C07161=1021.143,352.231,-144.972,171.488,49.524,159.785
C07162=1021.135,351.990,-144.936,171.480,49.525,159.784
C07163=1021.128,351.749,-144.900,171.473,49.527,159.783
C07164=1021.121,351.507,-144.863,171.466,49.529,159.782
C07165=1021.113,351.266,-144.827,171.459,49.530,159.781
C07166=1021.105,351.019,-144.788,171.451,49.531,159.781
C07167=1021.097,350.772,-144.751,171.444,49.532,159.780
C07168=1021.090,350.525,-144.714,171.437,49.534,159.779
C07169=1021.083,350.278,-144.676,171.429,49.535,159.778
C07170=1021.075,350.031,-144.639,171.422,49.536,159.777
C07171=1021.067,349.784,-144.602,171.416,49.538,159.777
C07172=1021.060,349.537,-144.565,171.408,49.539,159.776
C07173=1021.052,349.289,-144.528,171.400,49.541,159.775
C07174=1021.045,349.042,-144.490,171.393,49.542,159.774
C07175=1021.037,348.795,-144.454,171.386,49.543,159.773
C07176=1021.030,348.548,-144.416,171.379,49.545,159.772
C07177=1021.022,348.302,-144.379,171.371,49.546,159.772
C07178=1021.015,348.054,-144.342,171.364,49.548,159.771
C07179=1021.008,347.807,-144.305,171.357,49.549,159.770
C07180=1021.000,347.560,-144.268,171.350,49.551,159.769
C07181=1020.993,347.313,-144.230,171.343,49.552,159.768
C07182=1020.985,347.065,-144.194,171.336,49.554,159.768
C07183=1020.977,346.818,-144.157,171.329,49.555,159.767
C07184=1020.970,346.571,-144.120,171.321,49.557,159.766
C07185=1020.962,346.324,-144.083,171.314,49.559,159.765
C07186=1020.954,346.076,-144.047,171.308,49.560,159.765
C07187=1020.947,345.829,-144.010,171.300,49.562,159.764
C07188=1020.939,345.582,-143.973,171.293,49.564,159.763
C07189=1020.931,345.335,-143.936,171.286,49.565,159.763
C07190=1020.925,345.087,-143.900,171.279,49.567,159.762
C07191=1020.917,344.840,-143.863,171.272,49.568,159.761
C07192=1020.910,344.593,-143.826,171.265,49.570,159.760
C07193=1020.903,344.346,-143.790,171.258,49.571,159.760
C07194=1020.895,344.099,-143.753,171.250,49.573,159.759
C07195=1020.888,343.851,-143.716,171.244,49.574,159.758
C07196=1020.880,343.604,-143.680,171.237,49.577,159.758
C07197=1020.873,343.358,-143.644,171.230,49.578,159.757
C07198=1020.866,343.110,-143.607,171.223,49.580,159.756
C07199=1020.858,342.863,-143.571,171.216,49.581,159.755
C07200=1020.850,342.615,-143.534,171.208,49.583,159.755
C07201=1020.843,342.368,-143.498,171.202,49.585,159.754
C07202=1020.836,342.121,-143.461,171.195,49.587,159.753
C07203=1020.828,341.874,-143.425,171.189,49.588,159.753
C07204=1020.821,341.626,-143.388,171.182,49.591,159.752
C07205=1020.814,341.379,-143.352,171.174,49.592,159.751
C07206=1020.807,341.132,-143.316,171.168,49.594,159.751
C07207=1020.799,340.884,-143.280,171.161,49.596,159.750
C07208=1020.792,340.638,-143.244,171.154,49.597,159.749
C07209=1020.785,340.390,-143.207,171.147,49.600,159.749
C07210=1020.778,340.143,-143.171,171.140,49.601,159.748
C07211=1020.770,339.896,-143.135,171.134,49.603,159.747
C07212=1020.762,339.648,-143.099,171.127,49.605,159.747
C07213=1020.755,339.402,-143.063,171.120,49.606,159.746
C07214=1020.749,339.153,-143.027,171.113,49.609,159.745
C07215=1020.742,338.906,-142.991,171.106,49.611,159.745
C07216=1020.734,338.659,-142.955,171.100,49.612,159.744
C07217=1020.726,338.411,-142.918,171.093,49.615,159.744
C07218=1020.719,338.169,-142.883,171.086,49.616,159.743
C07219=1020.712,337.926,-142.848,171.079,49.618,159.742
C07220=1020.705,337.684,-142.814,171.073,49.620,159.742
C07221=1020.698,337.441,-142.778,171.066,49.622,159.741
C07222=1020.691,337.198,-142.743,171.060,49.624,159.741
C07223=1020.683,336.956,-142.708,171.054,49.626,159.740
C07224=1020.676,336.713,-142.673,171.047,49.628,159.740
C07225=1020.669,336.470,-142.638,171.040,49.630,159.739
C07226=1020.662,336.222,-142.602,171.033,49.632,159.738
C07227=1020.655,335.975,-142.566,171.027,49.634,159.738
C07228=1020.648,335.727,-142.531,171.020,49.636,159.737
C07229=1020.641,335.480,-142.495,171.014,49.638,159.737
C07230=1020.634,335.233,-142.460,171.007,49.641,159.736
C07231=1020.626,334.985,-142.424,171.001,49.642,159.736
C07232=1020.619,334.738,-142.388,170.994,49.644,159.735
C07233=1020.612,334.490,-142.353,170.988,49.646,159.734
C07234=1020.605,334.243,-142.317,170.981,49.649,159.734
C07235=1020.598,333.996,-142.282,170.975,49.651,159.733
C07236=1020.591,333.748,-142.246,170.968,49.653,159.733
C07237=1020.584,333.501,-142.211,170.962,49.655,159.732
C07238=1020.577,333.254,-142.176,170.955,49.657,159.732
C07239=1020.570,333.006,-142.140,170.949,49.659,159.731
C07240=1020.562,332.759,-142.105,170.942,49.662,159.731
C07241=1020.555,332.512,-142.070,170.936,49.664,159.730
C07242=1020.548,332.264,-142.034,170.929,49.666,159.730
C07243=1020.541,332.016,-141.999,170.923,49.668,159.729
C07244=1020.533,331.769,-141.964,170.916,49.670,159.729
C07245=1020.527,331.522,-141.929,170.910,49.673,159.728
C07246=1020.520,331.275,-141.894,170.903,49.675,159.728
C07247=1020.512,331.027,-141.859,170.897,49.677,159.727
C07248=1020.505,330.780,-141.824,170.890,49.680,159.727
C07249=1020.498,330.532,-141.789,170.884,49.681,159.726
C07250=1020.491,330.285,-141.754,170.877,49.684,159.726
C07251=1020.484,330.037,-141.718,170.871,49.686,159.725
C07252=1020.476,329.790,-141.684,170.864,49.689,159.725
C07253=1020.470,329.542,-141.649,170.858,49.691,159.724
C07254=1020.463,329.295,-141.614,170.851,49.694,159.724
C07255=1020.455,329.048,-141.579,170.845,49.696,159.723
C07256=1020.449,328.800,-141.545,170.838,49.698,159.723
C07257=1020.442,328.553,-141.509,170.833,49.701,159.723
C07258=1020.435,328.305,-141.474,170.826,49.703,159.722
C07259=1020.427,328.057,-141.439,170.820,49.706,159.722
C07260=1020.421,327.810,-141.404,170.814,49.708,159.721
C07261=1020.414,327.562,-141.370,170.807,49.710,159.721
C07262=1020.407,327.315,-141.335,170.801,49.713,159.720
C07263=1020.400,327.068,-141.300,170.794,49.715,159.720
C07264=1020.393,326.820,-141.265,170.789,49.718,159.719
C07265=1020.387,326.572,-141.231,170.782,49.720,159.719
C07266=1020.379,326.325,-141.196,170.776,49.723,159.719
C07267=1020.372,326.078,-141.162,170.769,49.725,159.718
C07268=1020.365,325.830,-141.127,170.763,49.727,159.718
C07269=1020.358,325.583,-141.093,170.758,49.730,159.717
C07270=1020.351,325.335,-141.059,170.751,49.733,159.717
C07271=1020.343,325.088,-141.025,170.745,49.735,159.717
C07272=1020.337,324.840,-140.991,170.738,49.738,159.716
C07273=1020.329,324.593,-140.956,170.733,49.741,159.716
C07274=1020.322,324.345,-140.922,170.726,49.744,159.715
C07275=1020.316,324.097,-140.888,170.720,49.746,159.715
C07276=1020.308,323.850,-140.853,170.713,49.749,159.715
C07277=1020.301,323.602,-140.819,170.708,49.751,159.714
C07278=1020.294,323.357,-140.786,170.701,49.754,159.714
C07279=1020.287,323.112,-140.752,170.695,49.757,159.714
C07280=1020.280,322.867,-140.718,170.689,49.759,159.713
C07281=1020.273,322.622,-140.685,170.683,49.762,159.713
C07282=1020.266,322.377,-140.650,170.677,49.764,159.712
C07283=1020.259,322.132,-140.617,170.671,49.767,159.712
C07284=1020.252,321.888,-140.583,170.665,49.770,159.712
C07285=1020.246,321.642,-140.549,170.659,49.773,159.712
C07286=1020.239,321.395,-140.516,170.653,49.775,159.711
C07287=1020.232,321.147,-140.482,170.647,49.778,159.711
C07288=1020.224,320.899,-140.448,170.641,49.781,159.711
C07289=1020.218,320.651,-140.414,170.634,49.784,159.710
C07290=1020.211,320.405,-140.379,170.629,49.787,159.710
C07291=1020.204,320.157,-140.346,170.623,49.789,159.710
C07292=1020.197,319.909,-140.311,170.616,49.792,159.709
C07293=1020.190,319.661,-140.277,170.611,49.795,159.709
C07294=1020.184,319.415,-140.244,170.604,49.798,159.709
C07295=1020.176,319.167,-140.210,170.598,49.800,159.708
C07296=1020.170,318.918,-140.176,170.593,49.803,159.708
C07297=1020.163,318.671,-140.142,170.586,49.806,159.708
C07298=1020.156,318.424,-140.109,170.580,49.809,159.707
C07299=1020.149,318.176,-140.075,170.574,49.812,159.707
C07300=1020.143,317.928,-140.041,170.568,49.814,159.707
C07301=1020.136,317.681,-140.007,170.563,49.818,159.706
C07302=1020.129,317.433,-139.973,170.556,49.821,159.706
C07303=1020.122,317.186,-139.940,170.551,49.823,159.706
C07304=1020.116,316.938,-139.906,170.545,49.826,159.705
C07305=1020.109,316.690,-139.872,170.538,49.829,159.705
C07306=1020.102,316.443,-139.839,170.533,49.832,159.705
C07307=1020.095,316.195,-139.805,170.527,49.835,159.705
C07308=1020.089,315.947,-139.771,170.521,49.838,159.704
C07309=1020.083,315.700,-139.738,170.515,49.840,159.704
C07310=1020.075,315.452,-139.704,170.510,49.844,159.704
C07311=1020.069,315.205,-139.671,170.503,49.847,159.704
C07312=1020.063,314.957,-139.637,170.497,49.849,159.703
C07313=1020.056,314.710,-139.604,170.492,49.853,159.703
C07314=1020.049,314.462,-139.570,170.485,49.855,159.703
C07315=1020.042,314.214,-139.537,170.480,49.858,159.702
C07316=1020.036,313.966,-139.503,170.474,49.861,159.702
C07317=1020.030,313.719,-139.470,170.468,49.864,159.702
C07318=1020.023,313.471,-139.436,170.462,49.867,159.702
C07319=1020.016,313.224,-139.403,170.457,49.870,159.702
C07320=1020.010,312.975,-139.369,170.451,49.873,159.701
C07321=1020.003,312.729,-139.335,170.445,49.877,159.701
C07322=1019.997,312.481,-139.303,170.439,49.879,159.701
C07323=1019.990,312.233,-139.269,170.434,49.883,159.701
C07324=1019.983,311.986,-139.236,170.427,49.886,159.700
C07325=1019.978,311.738,-139.202,170.422,49.889,159.700
C07326=1019.971,311.490,-139.169,170.416,49.891,159.700
C07327=1019.964,311.243,-139.135,170.411,49.895,159.700
C07328=1019.957,310.995,-139.102,170.404,49.898,159.699
C07329=1019.952,310.747,-139.069,170.399,49.901,159.699
C07330=1019.945,310.500,-139.036,170.393,49.904,159.699
C07331=1019.938,310.252,-139.002,170.388,49.907,159.699
C07332=1019.932,310.004,-138.970,170.382,49.910,159.699
C07333=1019.925,309.757,-138.936,170.376,49.913,159.698
C07334=1019.918,309.509,-138.903,170.371,49.917,159.698
C07335=1019.911,309.262,-138.871,170.365,49.920,159.698
C07336=1019.905,309.014,-138.838,170.359,49.923,159.698
C07337=1019.897,308.766,-138.806,170.353,49.927,159.698
C07338=1019.891,308.523,-138.774,170.347,49.930,159.698
C07339=1019.885,308.281,-138.742,170.342,49.933,159.697
C07340=1019.878,308.039,-138.710,170.337,49.936,159.697
C07341=1019.871,307.796,-138.678,170.332,49.940,159.697
C07342=1019.864,307.553,-138.647,170.325,49.943,159.697
C07343=1019.858,307.311,-138.615,170.320,49.947,159.697
C07344=1019.852,307.069,-138.582,170.315,49.950,159.697
C07345=1019.845,306.827,-138.551,170.309,49.953,159.697
C07346=1019.839,306.579,-138.519,170.303,49.957,159.697
C07347=1019.831,306.331,-138.486,170.298,49.960,159.696
C07348=1019.825,306.083,-138.453,170.293,49.963,159.696
C07349=1019.819,305.836,-138.421,170.286,49.967,159.696
C07350=1019.812,305.588,-138.389,170.281,49.970,159.696
C07351=1019.806,305.340,-138.357,170.276,49.974,159.696
C07352=1019.798,305.092,-138.324,170.269,49.977,159.696
C07353=1019.792,304.845,-138.291,170.264,49.981,159.696
C07354=1019.785,304.597,-138.259,170.259,49.984,159.696
C07355=1019.779,304.349,-138.227,170.253,49.987,159.695
C07356=1019.772,304.102,-138.194,170.247,49.991,159.695
C07357=1019.765,303.854,-138.162,170.242,49.995,159.695
C07358=1019.759,303.605,-138.130,170.236,49.998,159.695
C07359=1019.752,303.358,-138.097,170.231,50.002,159.695
C07360=1019.745,303.110,-138.065,170.226,50.005,159.695
C07361=1019.739,302.862,-138.033,170.219,50.009,159.695
C07362=1019.732,302.615,-138.001,170.214,50.013,159.695
C07363=1019.726,302.367,-137.969,170.209,50.016,159.695
C07364=1019.719,302.119,-137.937,170.204,50.019,159.695
C07365=1019.713,301.872,-137.904,170.198,50.023,159.694
C07366=1019.707,301.624,-137.872,170.192,50.026,159.694
C07367=1019.699,301.376,-137.839,170.187,50.030,159.694
C07368=1019.693,301.127,-137.807,170.181,50.034,159.694
C07369=1019.686,300.880,-137.775,170.176,50.037,159.694
C07370=1019.680,300.632,-137.743,170.171,50.041,159.694
C07371=1019.674,300.384,-137.712,170.165,50.045,159.694
C07372=1019.667,300.136,-137.679,170.159,50.048,159.694
C07373=1019.661,299.888,-137.647,170.154,50.052,159.694
C07374=1019.654,299.641,-137.615,170.149,50.055,159.694
C07375=1019.648,299.393,-137.583,170.143,50.059,159.694
C07376=1019.641,299.145,-137.551,170.138,50.063,159.694
C07377=1019.635,298.897,-137.519,170.133,50.066,159.694
C07378=1019.629,298.650,-137.487,170.128,50.070,159.694
C07379=1019.623,298.402,-137.455,170.121,50.074,159.694
C07380=1019.617,298.154,-137.423,170.116,50.077,159.693
C07381=1019.610,297.906,-137.391,170.111,50.081,159.694
C07382=1019.604,297.658,-137.359,170.106,50.084,159.693
C07383=1019.597,297.411,-137.327,170.100,50.089,159.693
C07384=1019.591,297.163,-137.295,170.095,50.092,159.693
C07385=1019.585,296.915,-137.264,170.090,50.096,159.693
C07386=1019.579,296.667,-137.232,170.084,50.100,159.693
C07387=1019.572,296.419,-137.199,170.079,50.104,159.693
C07388=1019.566,296.172,-137.168,170.073,50.107,159.693
C07389=1019.560,295.924,-137.136,170.069,50.111,159.693
C07390=1019.553,295.676,-137.104,170.063,50.115,159.693
C07391=1019.547,295.427,-137.072,170.057,50.118,159.693
C07392=1019.541,295.179,-137.041,170.052,50.122,159.693
C07393=1019.535,294.933,-137.009,170.047,50.126,159.693
C07394=1019.529,294.684,-136.976,170.042,50.130,159.693
C07395=1019.522,294.436,-136.945,170.036,50.134,159.693
C07396=1019.516,294.188,-136.913,170.031,50.137,159.693
C07397=1019.510,293.940,-136.882,170.026,50.141,159.693
C07398=1019.504,293.707,-136.853,170.021,50.145,159.693
C07399=1019.499,293.473,-136.822,170.016,50.149,159.693
C07400=1019.492,293.240,-136.792,170.011,50.152,159.693
C07401=1019.486,293.006,-136.762,170.006,50.156,159.693
C07402=1019.481,292.772,-136.733,170.001,50.160,159.693
C07403=1019.475,292.539,-136.703,169.996,50.163,159.693
C07404=1019.469,292.305,-136.674,169.992,50.167,159.693
C07405=1019.462,292.072,-136.644,169.987,50.171,159.693
C07406=1019.457,291.823,-136.613,169.981,50.175,159.693
C07407=1019.450,291.575,-136.582,169.976,50.179,159.694
C07408=1019.443,291.328,-136.550,169.971,50.183,159.694
C07409=1019.437,291.080,-136.519,169.965,50.187,159.694
C07410=1019.431,290.832,-136.488,169.960,50.191,159.694
C07411=1019.424,290.584,-136.457,169.955,50.195,159.694
C07412=1019.419,290.336,-136.426,169.951,50.199,159.694
C07413=1019.412,290.088,-136.395,169.945,50.204,159.694
C07414=1019.405,289.840,-136.363,169.940,50.208,159.694
C07415=1019.400,289.592,-136.333,169.935,50.212,159.694
C07416=1019.393,289.344,-136.301,169.929,50.216,159.694
C07417=1019.386,289.096,-136.271,169.924,50.220,159.694
C07418=1019.380,288.849,-136.240,169.919,50.224,159.694
C07419=1019.374,288.601,-136.208,169.913,50.228,159.694
C07420=1019.367,288.352,-136.177,169.908,50.232,159.694
C07421=1019.361,288.105,-136.146,169.903,50.236,159.694
C07422=1019.355,287.856,-136.116,169.899,50.240,159.694
C07423=1019.348,287.608,-136.084,169.893,50.245,159.694
C07424=1019.342,287.361,-136.054,169.888,50.249,159.695
C07425=1019.336,287.112,-136.023,169.883,50.253,159.695
C07426=1019.329,286.865,-135.992,169.877,50.258,159.695
C07427=1019.323,286.616,-135.961,169.872,50.262,159.695
C07428=1019.316,286.369,-135.930,169.868,50.265,159.695
C07429=1019.311,286.121,-135.900,169.863,50.270,159.695
C07430=1019.304,285.872,-135.869,169.857,50.274,159.695
C07431=1019.298,285.625,-135.838,169.852,50.278,159.695
C07432=1019.292,285.376,-135.807,169.847,50.282,159.695
C07433=1019.286,285.129,-135.777,169.842,50.287,159.696
C07434=1019.279,284.881,-135.745,169.837,50.291,159.696
C07435=1019.273,284.633,-135.715,169.832,50.295,159.696
C07436=1019.267,284.384,-135.684,169.827,50.300,159.696
C07437=1019.261,284.137,-135.654,169.822,50.304,159.696
C07438=1019.255,283.888,-135.623,169.817,50.309,159.696
C07439=1019.248,283.641,-135.593,169.811,50.313,159.696
C07440=1019.242,283.392,-135.563,169.807,50.318,159.697
C07441=1019.235,283.145,-135.532,169.802,50.322,159.697
C07442=1019.229,282.896,-135.501,169.796,50.327,159.697
C07443=1019.222,282.649,-135.471,169.791,50.331,159.697
C07444=1019.216,282.400,-135.440,169.787,50.336,159.697
C07445=1019.210,282.152,-135.410,169.782,50.340,159.697
C07446=1019.204,281.904,-135.379,169.776,50.345,159.698
C07447=1019.197,281.656,-135.350,169.772,50.349,159.698
C07448=1019.191,281.409,-135.319,169.767,50.353,159.698
C07449=1019.185,281.160,-135.289,169.761,50.358,159.698
C07450=1019.179,280.912,-135.258,169.757,50.362,159.698
C07451=1019.173,280.664,-135.228,169.752,50.366,159.698
C07452=1019.166,280.416,-135.198,169.746,50.371,159.698
C07453=1019.160,280.168,-135.167,169.742,50.376,159.699
C07454=1019.154,279.920,-135.137,169.737,50.380,159.699
C07455=1019.148,279.671,-135.107,169.731,50.385,159.699
C07456=1019.141,279.423,-135.077,169.726,50.389,159.699
C07457=1019.136,279.175,-135.047,169.722,50.394,159.699
C07458=1019.130,278.948,-135.019,169.717,50.398,159.699
C07459=1019.124,278.721,-134.991,169.713,50.402,159.700
C07460=1019.119,278.493,-134.963,169.708,50.406,159.700
C07461=1019.113,278.265,-134.936,169.704,50.411,159.700
C07462=1019.108,278.038,-134.908,169.699,50.415,159.700
C07463=1019.102,277.810,-134.880,169.694,50.419,159.700
C07464=1019.096,277.583,-134.852,169.690,50.423,159.701
C07465=1019.090,277.355,-134.825,169.685,50.427,159.701
C07466=1019.084,277.107,-134.795,169.681,50.432,159.701
C07467=1019.079,276.859,-134.765,169.676,50.437,159.701
C07468=1019.073,276.611,-134.734,169.672,50.441,159.702
C07469=1019.066,276.363,-134.705,169.666,50.446,159.702
C07470=1019.060,276.115,-134.674,169.661,50.450,159.702
C07471=1019.054,275.867,-134.645,169.657,50.455,159.702
C07472=1019.047,275.618,-134.615,169.651,50.460,159.702
C07473=1019.041,275.371,-134.585,169.647,50.465,159.703
C07474=1019.035,275.122,-134.555,169.641,50.470,159.703
C07475=1019.029,274.875,-134.525,169.637,50.475,159.703
C07476=1019.023,274.626,-134.495,169.632,50.479,159.703
C07477=1019.016,274.378,-134.466,169.627,50.484,159.704
C07478=1019.011,274.130,-134.436,169.622,50.489,159.704
C07479=1019.004,273.882,-134.406,169.618,50.494,159.704
C07480=1018.999,273.634,-134.377,169.612,50.499,159.704
C07481=1018.991,273.385,-134.347,169.608,50.503,159.705
C07482=1018.986,273.137,-134.317,169.603,50.508,159.705
C07483=1018.979,272.889,-134.287,169.598,50.513,159.705
C07484=1018.974,272.641,-134.258,169.593,50.518,159.705
C07485=1018.968,272.393,-134.229,169.589,50.522,159.706
C07486=1018.962,272.145,-134.198,169.583,50.527,159.706
C07487=1018.955,271.896,-134.169,169.579,50.532,159.706
C07488=1018.949,271.648,-134.140,169.575,50.537,159.707
C07489=1018.943,271.400,-134.109,169.569,50.542,159.707
C07490=1018.937,271.152,-134.080,169.565,50.547,159.707
C07491=1018.931,270.904,-134.051,169.560,50.552,159.707
C07492=1018.925,270.656,-134.021,169.555,50.557,159.707
C07493=1018.918,270.408,-133.992,169.550,50.562,159.708
C07494=1018.913,270.160,-133.962,169.545,50.567,159.708
C07495=1018.906,269.911,-133.933,169.540,50.572,159.708
C07496=1018.900,269.662,-133.903,169.536,50.577,159.709
C07497=1018.894,269.415,-133.873,169.530,50.582,159.709
C07498=1018.888,269.167,-133.844,169.526,50.587,159.709
C07499=1018.882,268.918,-133.815,169.522,50.592,159.710
C07500=1018.876,268.670,-133.786,169.516,50.597,159.710
C07501=1018.870,268.422,-133.757,169.512,50.602,159.710
C07502=1018.863,268.174,-133.728,169.507,50.607,159.710
C07503=1018.858,267.925,-133.698,169.502,50.612,159.711
C07504=1018.852,267.677,-133.669,169.498,50.617,159.711
C07505=1018.845,267.429,-133.640,169.493,50.622,159.711
C07506=1018.839,267.181,-133.611,169.488,50.627,159.712
C07507=1018.834,266.933,-133.581,169.484,50.632,159.712
C07508=1018.827,266.684,-133.552,169.479,50.637,159.712
C07509=1018.821,266.436,-133.523,169.474,50.643,159.713
C07510=1018.815,266.188,-133.494,169.469,50.648,159.713
C07511=1018.809,265.940,-133.465,169.465,50.653,159.714
C07512=1018.803,265.692,-133.435,169.460,50.658,159.714
C07513=1018.797,265.443,-133.406,169.455,50.664,159.714
C07514=1018.791,265.195,-133.377,169.451,50.668,159.714
C07515=1018.784,264.947,-133.348,169.446,50.674,159.715
C07516=1018.778,264.699,-133.319,169.441,50.679,159.715
C07517=1018.772,264.451,-133.290,169.437,50.684,159.716
C07518=1018.767,264.226,-133.264,169.433,50.689,159.716
C07519=1018.762,264.000,-133.238,169.428,50.693,159.716
C07520=1018.755,263.775,-133.212,169.424,50.698,159.716
C07521=1018.750,263.550,-133.185,169.419,50.703,159.717
C07522=1018.745,263.324,-133.159,169.415,50.708,159.717
C07523=1018.739,263.099,-133.134,169.412,50.713,159.718
C07524=1018.734,262.875,-133.107,169.407,50.717,159.718
C07525=1018.728,262.649,-133.081,169.403,50.722,159.718
C07526=1018.722,262.400,-133.052,169.398,50.728,159.718
C07527=1018.717,262.153,-133.023,169.393,50.733,159.719
C07528=1018.710,261.904,-132.994,169.389,50.738,159.719
C07529=1018.704,261.656,-132.966,169.384,50.744,159.720
C07530=1018.698,261.408,-132.937,169.380,50.749,159.720
C07531=1018.692,261.159,-132.907,169.375,50.755,159.720
C07532=1018.686,260.911,-132.879,169.370,50.759,159.721
C07533=1018.680,260.662,-132.850,169.366,50.765,159.721
C07534=1018.674,260.415,-132.821,169.361,50.771,159.722
C07535=1018.668,260.166,-132.793,169.357,50.776,159.722
C07536=1018.662,259.918,-132.764,169.352,50.781,159.722
C07537=1018.656,259.669,-132.736,169.347,50.786,159.723
C07538=1018.649,259.422,-132.707,169.342,50.792,159.723
C07539=1018.643,259.173,-132.679,169.338,50.798,159.724
C07540=1018.638,258.925,-132.651,169.333,50.803,159.724
C07541=1018.631,258.677,-132.623,169.329,50.809,159.724
C07542=1018.625,258.428,-132.594,169.324,50.814,159.725
C07543=1018.619,258.179,-132.566,169.320,50.820,159.725
C07544=1018.612,257.932,-132.537,169.315,50.826,159.726
C07545=1018.606,257.683,-132.509,169.311,50.832,159.726
C07546=1018.601,257.435,-132.481,169.306,50.837,159.727
C07547=1018.594,257.187,-132.453,169.301,50.843,159.727
C07548=1018.588,256.938,-132.424,169.297,50.848,159.728
C07549=1018.582,256.690,-132.396,169.292,50.854,159.728
C07550=1018.575,256.441,-132.368,169.288,50.860,159.729
C07551=1018.570,256.193,-132.340,169.283,50.865,159.729
C07552=1018.563,255.945,-132.311,169.279,50.871,159.729
C07553=1018.557,255.696,-132.284,169.273,50.877,159.730
C07554=1018.551,255.448,-132.255,169.269,50.882,159.730
C07555=1018.545,255.200,-132.227,169.265,50.888,159.731
C07556=1018.539,254.951,-132.200,169.261,50.894,159.731
C07557=1018.533,254.703,-132.171,169.256,50.900,159.732
C07558=1018.527,254.455,-132.143,169.252,50.905,159.732
C07559=1018.521,254.207,-132.115,169.246,50.911,159.733
C07560=1018.515,253.958,-132.087,169.243,50.917,159.733
C07561=1018.508,253.709,-132.059,169.238,50.923,159.734
C07562=1018.503,253.461,-132.031,169.234,50.928,159.734
C07563=1018.497,253.213,-132.003,169.229,50.934,159.734
C07564=1018.490,252.964,-131.975,169.224,50.940,159.735
C07565=1018.485,252.716,-131.947,169.220,50.946,159.736
C07566=1018.479,252.467,-131.919,169.215,50.951,159.736
C07567=1018.472,252.220,-131.890,169.211,50.957,159.736
C07568=1018.466,251.972,-131.862,169.206,50.963,159.737
C07569=1018.460,251.723,-131.834,169.202,50.969,159.737
C07570=1018.454,251.475,-131.806,169.197,50.974,159.738
C07571=1018.448,251.226,-131.778,169.193,50.980,159.738
C07572=1018.442,250.977,-131.750,169.188,50.986,159.739
C07573=1018.436,250.730,-131.722,169.184,50.992,159.739
C07574=1018.431,250.480,-131.695,169.179,50.998,159.740
C07575=1018.425,250.233,-131.667,169.175,51.003,159.740
C07576=1018.419,249.984,-131.639,169.171,51.010,159.741
C07577=1018.413,249.735,-131.611,169.167,51.015,159.741
C07578=1018.407,249.510,-131.586,169.163,51.021,159.742
C07579=1018.402,249.284,-131.560,169.158,51.026,159.742
C07580=1018.396,249.057,-131.535,169.154,51.032,159.743
C07581=1018.392,248.831,-131.509,169.150,51.037,159.743
C07582=1018.386,248.605,-131.484,169.146,51.042,159.744
C07583=1018.381,248.379,-131.459,169.142,51.048,159.744
C07584=1018.375,248.154,-131.434,169.138,51.053,159.745
C07585=1018.370,247.927,-131.408,169.134,51.059,159.745
C07586=1018.364,247.679,-131.380,169.129,51.065,159.746
C07587=1018.358,247.430,-131.353,169.125,51.071,159.746
C07588=1018.353,247.182,-131.325,169.120,51.076,159.747
C07589=1018.346,246.934,-131.297,169.117,51.083,159.747
C07590=1018.341,246.685,-131.269,169.112,51.088,159.748
C07591=1018.334,246.437,-131.241,169.108,51.094,159.748
C07592=1018.329,246.188,-131.214,169.103,51.100,159.749
C07593=1018.323,245.940,-131.186,169.098,51.107,159.749
C07594=1018.317,245.692,-131.158,169.094,51.112,159.750
C07595=1018.311,245.443,-131.131,169.090,51.119,159.750
C07596=1018.306,245.194,-131.103,169.085,51.124,159.751
C07597=1018.300,244.947,-131.075,169.081,51.130,159.751
C07598=1018.294,244.698,-131.047,169.077,51.137,159.752
C07599=1018.288,244.450,-131.021,169.072,51.142,159.753
C07600=1018.282,244.201,-130.992,169.068,51.148,159.753
C07601=1018.277,243.953,-130.964,169.064,51.155,159.754
C07602=1018.271,243.704,-130.938,169.060,51.160,159.754
C07603=1018.265,243.456,-130.909,169.055,51.167,159.755
C07604=1018.259,243.208,-130.882,169.050,51.173,159.755
C07605=1018.254,242.959,-130.854,169.046,51.179,159.756
C07606=1018.247,242.711,-130.827,169.042,51.185,159.756
C07607=1018.242,242.462,-130.800,169.038,51.191,159.757
C07608=1018.236,242.214,-130.772,169.034,51.198,159.758
C07609=1018.230,241.965,-130.745,169.029,51.204,159.758
C07610=1018.222,241.657,-130.711,169.024,51.212,159.759
C07611=1018.216,241.348,-130.677,169.018,51.219,159.760
C07612=1018.208,241.040,-130.643,169.014,51.227,159.761
C07613=1018.201,240.731,-130.610,169.007,51.235,159.761
C07614=1018.195,240.483,-130.582,169.004,51.241,159.762
C07615=1018.189,240.233,-130.555,168.999,51.248,159.762
C07616=1018.183,239.985,-130.528,168.994,51.254,159.763
C07617=1018.177,239.737,-130.501,168.991,51.261,159.764
C07618=1018.172,239.489,-130.474,168.986,51.267,159.764
C07619=1018.166,239.240,-130.447,168.981,51.274,159.765
C07620=1018.160,238.992,-130.419,168.978,51.280,159.766
C07621=1018.154,238.743,-130.393,168.973,51.286,159.766
C07622=1018.148,238.494,-130.366,168.969,51.293,159.767
C07623=1018.143,238.246,-130.338,168.965,51.299,159.767
C07624=1018.137,237.998,-130.311,168.960,51.305,159.768
C07625=1018.130,237.749,-130.284,168.956,51.312,159.769
C07626=1018.124,237.501,-130.257,168.951,51.318,159.769
C07627=1018.119,237.252,-130.231,168.947,51.324,159.770
C07628=1018.113,237.004,-130.204,168.943,51.332,159.771
C07629=1018.107,236.755,-130.177,168.939,51.338,159.771
C07630=1018.101,236.506,-130.150,168.934,51.345,159.772
C07631=1018.095,236.258,-130.124,168.930,51.351,159.772
C07632=1018.089,236.010,-130.097,168.926,51.357,159.773
C07633=1018.083,235.761,-130.069,168.921,51.364,159.774
C07634=1018.077,235.513,-130.043,168.918,51.371,159.775
C07635=1018.071,235.265,-130.016,168.913,51.377,159.775
C07636=1018.065,235.016,-129.989,168.909,51.384,159.776
C07637=1018.059,234.767,-129.962,168.904,51.391,159.776
C07638=1018.049,234.368,-129.920,168.897,51.401,159.777
C07639=1018.040,233.970,-129.876,168.891,51.412,159.779
C07640=1018.031,233.571,-129.834,168.884,51.422,159.780
C07641=1018.022,233.173,-129.792,168.877,51.433,159.781
C07642=1018.015,232.924,-129.765,168.873,51.440,159.781
C07643=1018.010,232.676,-129.739,168.868,51.447,159.782
C07644=1018.004,232.428,-129.712,168.865,51.453,159.783
C07645=1017.998,232.179,-129.685,168.861,51.460,159.784
C07646=1017.992,231.931,-129.659,168.856,51.466,159.784
C07647=1017.986,231.682,-129.632,168.852,51.474,159.785
C07648=1017.981,231.434,-129.605,168.847,51.480,159.785
C07649=1017.975,231.184,-129.579,168.844,51.487,159.786
C07650=1017.969,230.936,-129.552,168.839,51.494,159.787
C07651=1017.963,230.688,-129.526,168.835,51.500,159.788
C07652=1017.957,230.439,-129.499,168.831,51.507,159.788
C07653=1017.952,230.191,-129.472,168.826,51.514,159.789
C07654=1017.946,229.942,-129.447,168.823,51.521,159.790
C07655=1017.940,229.694,-129.420,168.818,51.527,159.790
C07656=1017.935,229.445,-129.393,168.814,51.534,159.791
C07657=1017.929,229.197,-129.367,168.810,51.542,159.792
C07658=1017.923,228.948,-129.341,168.805,51.548,159.792
C07659=1017.917,228.700,-129.315,168.802,51.555,159.793
C07660=1017.911,228.452,-129.288,168.797,51.562,159.794
C07661=1017.906,228.203,-129.262,168.793,51.569,159.795
C07662=1017.899,227.953,-129.235,168.789,51.576,159.796
C07663=1017.893,227.705,-129.208,168.784,51.582,159.796
C07664=1017.887,227.456,-129.183,168.780,51.590,159.797
C07665=1017.881,227.208,-129.156,168.776,51.597,159.798
C07666=1017.876,226.959,-129.130,168.772,51.603,159.798
C07667=1017.870,226.711,-129.104,168.768,51.610,159.799
C07668=1017.864,226.462,-129.077,168.764,51.618,159.800
C07669=1017.858,226.214,-129.052,168.760,51.625,159.801
C07670=1017.852,225.965,-129.025,168.756,51.632,159.802
C07671=1017.846,225.717,-129.000,168.751,51.639,159.802
C07672=1017.841,225.468,-128.974,168.747,51.646,159.803
C07673=1017.835,225.219,-128.947,168.743,51.653,159.804
C07674=1017.829,224.971,-128.922,168.739,51.660,159.804
C07675=1017.823,224.722,-128.895,168.734,51.667,159.805
C07676=1017.817,224.474,-128.870,168.730,51.675,159.806
C07677=1017.811,224.225,-128.844,168.726,51.682,159.807
C07678=1017.806,223.976,-128.817,168.723,51.689,159.808
C07679=1017.799,223.728,-128.792,168.719,51.696,159.809
C07680=1017.794,223.479,-128.766,168.714,51.703,159.809
C07681=1017.788,223.231,-128.740,168.710,51.710,159.810
C07682=1017.782,222.982,-128.714,168.706,51.717,159.811
C07683=1017.776,222.734,-128.689,168.702,51.724,159.811
C07684=1017.771,222.485,-128.662,168.698,51.732,159.812
C07685=1017.765,222.236,-128.637,168.693,51.739,159.813
C07686=1017.759,221.988,-128.611,168.689,51.746,159.814
C07687=1017.753,221.739,-128.585,168.685,51.753,159.815
C07688=1017.747,221.491,-128.559,168.681,51.761,159.815
C07689=1017.741,221.242,-128.533,168.677,51.768,159.816
C07690=1017.735,220.993,-128.508,168.673,51.775,159.817
C07691=1017.729,220.745,-128.481,168.669,51.783,159.818
C07692=1017.725,220.496,-128.456,168.665,51.790,159.819
C07693=1017.718,220.248,-128.430,168.661,51.798,159.820
C07694=1017.712,220.014,-128.406,168.657,51.804,159.820
C07695=1017.707,219.781,-128.382,168.653,51.811,159.821
C07696=1017.702,219.548,-128.358,168.649,51.818,159.822
C07697=1017.697,219.313,-128.333,168.645,51.824,159.822
C07698=1017.691,219.080,-128.309,168.641,51.832,159.823
C07699=1017.686,218.847,-128.285,168.638,51.839,159.824
C07700=1017.681,218.613,-128.261,168.633,51.845,159.825
C07701=1017.675,218.379,-128.236,168.630,51.852,159.826
C07702=1017.669,218.131,-128.210,168.626,51.859,159.826
C07703=1017.664,217.883,-128.185,168.622,51.867,159.827
C07704=1017.657,217.634,-128.160,168.617,51.875,159.828
C07705=1017.651,217.385,-128.135,168.613,51.882,159.829
C07706=1017.646,217.136,-128.109,168.609,51.890,159.830
C07707=1017.640,216.888,-128.084,168.605,51.897,159.831
C07708=1017.634,216.640,-128.058,168.601,51.905,159.831
C07709=1017.628,216.391,-128.033,168.597,51.913,159.832
C07710=1017.622,216.142,-128.007,168.593,51.920,159.833
C07711=1017.616,215.893,-127.982,168.589,51.927,159.834
C07712=1017.610,215.645,-127.957,168.585,51.935,159.835
C07713=1017.605,215.396,-127.932,168.581,51.942,159.836
C07714=1017.599,215.147,-127.906,168.576,51.951,159.837
C07715=1017.593,214.898,-127.881,168.572,51.958,159.838
C07716=1017.587,214.650,-127.856,168.569,51.966,159.839
C07717=1017.582,214.401,-127.830,168.565,51.973,159.839
C07718=1017.576,214.153,-127.805,168.561,51.981,159.840
C07719=1017.569,213.904,-127.779,168.557,51.989,159.841
C07720=1017.564,213.656,-127.754,168.553,51.996,159.842
C07721=1017.559,213.407,-127.729,168.549,52.004,159.843
C07722=1017.552,213.158,-127.704,168.544,52.012,159.844
C07723=1017.546,212.909,-127.679,168.540,52.019,159.845
C07724=1017.541,212.661,-127.653,168.536,52.027,159.846
C07725=1017.535,212.412,-127.628,168.532,52.035,159.846
C07726=1017.529,212.163,-127.603,168.529,52.043,159.847
C07727=1017.524,211.915,-127.578,168.524,52.050,159.848
C07728=1017.518,211.666,-127.552,168.521,52.058,159.849
C07729=1017.512,211.417,-127.527,168.516,52.066,159.850
C07730=1017.507,211.169,-127.503,168.512,52.074,159.851
C07731=1017.500,210.920,-127.477,168.508,52.082,159.852
C07732=1017.495,210.671,-127.451,168.504,52.089,159.853
C07733=1017.489,210.423,-127.426,168.500,52.097,159.854
C07734=1017.483,210.174,-127.402,168.496,52.104,159.854
C07735=1017.477,209.925,-127.376,168.493,52.112,159.855
C07736=1017.472,209.677,-127.351,168.488,52.121,159.856
C07737=1017.466,209.428,-127.326,168.484,52.128,159.857
C07738=1017.461,209.180,-127.301,168.480,52.136,159.858
C07739=1017.455,208.930,-127.277,168.477,52.144,159.859
C07740=1017.449,208.682,-127.251,168.472,52.152,159.860
C07741=1017.443,208.434,-127.226,168.468,52.160,159.861
C07742=1017.437,208.184,-127.202,168.464,52.168,159.862
C07743=1017.431,207.936,-127.176,168.460,52.176,159.863
C07744=1017.426,207.687,-127.152,168.456,52.184,159.864
C07745=1017.420,207.438,-127.127,168.452,52.192,159.865
C07746=1017.414,207.190,-127.102,168.448,52.200,159.866
C07747=1017.408,206.941,-127.077,168.445,52.208,159.867
C07748=1017.403,206.693,-127.053,168.440,52.216,159.868
C07749=1017.397,206.444,-127.028,168.436,52.224,159.868
C07750=1017.391,206.195,-127.003,168.432,52.232,159.869
C07751=1017.385,205.947,-126.978,168.429,52.240,159.870
C07752=1017.379,205.697,-126.953,168.424,52.248,159.871
C07753=1017.374,205.449,-126.929,168.420,52.256,159.872
C07754=1017.369,205.212,-126.905,168.417,52.264,159.873
C07755=1017.362,204.975,-126.882,168.413,52.271,159.874
C07756=1017.357,204.739,-126.859,168.409,52.280,159.875
C07757=1017.352,204.503,-126.836,168.405,52.288,159.876
C07758=1017.346,204.265,-126.812,168.401,52.295,159.877
C07759=1017.340,204.029,-126.789,168.398,52.303,159.878
C07760=1017.335,203.793,-126.765,168.394,52.311,159.879
C07761=1017.330,203.556,-126.742,168.390,52.319,159.880
C07762=1017.305,202.315,-126.626,167.903,52.236,159.767
C07763=1017.300,202.066,-126.604,167.898,52.246,159.768
C07764=1017.296,201.818,-126.581,167.894,52.255,159.769
C07765=1017.291,201.570,-126.558,167.889,52.264,159.770
C07766=1017.286,201.321,-126.535,167.884,52.273,159.771
C07767=1017.281,201.072,-126.513,167.880,52.282,159.772
C07768=1017.276,200.823,-126.489,167.875,52.291,159.773
C07769=1017.272,200.573,-126.467,167.870,52.301,159.774
C07770=1017.267,200.325,-126.444,167.866,52.310,159.775
C07771=1017.262,200.077,-126.421,167.861,52.319,159.776
C07772=1017.257,199.827,-126.398,167.857,52.329,159.778
C07773=1017.253,199.578,-126.375,167.852,52.338,159.779
C07774=1017.248,199.329,-126.353,167.848,52.348,159.780
C07775=1017.243,199.080,-126.329,167.843,52.357,159.781
C07776=1017.238,198.831,-126.307,167.838,52.366,159.782
C07777=1017.233,198.583,-126.285,167.834,52.376,159.783
C07778=1017.229,198.333,-126.262,167.829,52.385,159.784
C07779=1017.223,198.085,-126.239,167.825,52.395,159.785
C07780=1017.218,197.836,-126.217,167.820,52.405,159.786
C07781=1017.214,197.587,-126.195,167.816,52.414,159.787
C07782=1017.208,197.338,-126.172,167.811,52.423,159.788
C07783=1017.203,197.089,-126.150,167.806,52.433,159.789
C07784=1017.199,196.840,-126.128,167.802,52.442,159.790
C07785=1017.194,196.591,-126.105,167.797,52.452,159.791
C07786=1017.189,196.342,-126.083,167.793,52.461,159.792
C07787=1017.184,196.093,-126.061,167.789,52.471,159.794
C07788=1017.179,195.844,-126.037,167.784,52.480,159.795
C07789=1017.174,195.595,-126.015,167.780,52.490,159.796
C07790=1017.169,195.346,-125.994,167.776,52.499,159.797
C07791=1017.165,195.097,-125.971,167.770,52.509,159.798
C07792=1017.159,194.848,-125.948,167.766,52.518,159.799
C07793=1017.155,194.600,-125.926,167.762,52.528,159.800
C07794=1017.151,194.350,-125.904,167.757,52.537,159.801
C07795=1017.145,194.101,-125.882,167.753,52.547,159.802
C07796=1017.140,193.853,-125.859,167.749,52.557,159.803
C07797=1017.135,193.604,-125.837,167.744,52.566,159.804
C07798=1017.131,193.355,-125.815,167.739,52.575,159.805
C07799=1017.126,193.105,-125.793,167.736,52.585,159.807
C07800=1017.121,192.856,-125.771,167.730,52.595,159.807
C07801=1017.117,192.607,-125.748,167.726,52.604,159.809
C07802=1017.112,192.359,-125.726,167.722,52.613,159.810
C07803=1017.106,192.110,-125.703,167.718,52.623,159.811
C07804=1017.101,191.861,-125.682,167.713,52.632,159.812
C07805=1017.097,191.612,-125.659,167.709,52.642,159.813
C07806=1017.092,191.363,-125.637,167.705,52.651,159.814
C07807=1017.088,191.114,-125.615,167.701,52.661,159.815
C07808=1017.083,190.864,-125.593,167.695,52.670,159.816
C07809=1017.078,190.615,-125.571,167.692,52.680,159.817
C07810=1017.073,190.367,-125.548,167.687,52.689,159.818
C07811=1017.069,190.118,-125.526,167.683,52.698,159.819
C07812=1017.064,189.869,-125.504,167.678,52.709,159.821
C07813=1017.059,189.620,-125.482,167.674,52.718,159.822
C07814=1017.054,189.372,-125.460,167.670,52.727,159.823
C07815=1017.050,189.122,-125.437,167.666,52.737,159.824
C07816=1017.045,188.873,-125.415,167.661,52.747,159.825
C07817=1017.040,188.624,-125.393,167.657,52.756,159.826
C07818=1017.035,188.375,-125.372,167.653,52.766,159.827
C07819=1017.031,188.126,-125.349,167.649,52.775,159.828
C07820=1017.026,187.877,-125.327,167.645,52.784,159.829
C07821=1017.022,187.629,-125.305,167.640,52.794,159.830
C07822=1017.017,187.348,-125.280,167.635,52.805,159.832
C07823=1017.011,187.068,-125.255,167.631,52.816,159.833
C07824=1017.007,186.787,-125.231,167.626,52.826,159.834
C07825=1017.001,186.507,-125.206,167.622,52.837,159.836
C07826=1016.996,186.258,-125.185,167.616,52.847,159.836
C07827=1016.992,186.009,-125.163,167.612,52.856,159.838
C07828=1016.987,185.760,-125.140,167.608,52.866,159.839
C07829=1016.983,185.511,-125.119,167.604,52.875,159.840
C07830=1016.978,185.262,-125.097,167.600,52.884,159.841
C07831=1016.974,185.013,-125.074,167.596,52.894,159.842
C07832=1016.969,184.764,-125.052,167.592,52.903,159.843
C07833=1016.964,184.516,-125.030,167.588,52.913,159.844
C07834=1016.959,184.267,-125.009,167.583,52.923,159.845
C07835=1016.955,184.017,-124.987,167.579,52.932,159.846
C07836=1016.951,183.768,-124.965,167.575,52.941,159.847
C07837=1016.946,183.519,-124.943,167.571,52.951,159.849
C07838=1016.941,183.270,-124.921,167.567,52.961,159.850
C07839=1016.937,183.021,-124.899,167.563,52.970,159.851
C07840=1016.932,182.772,-124.878,167.559,52.980,159.852
C07841=1016.928,182.523,-124.856,167.555,52.989,159.853
C07842=1016.924,182.274,-124.833,167.551,52.998,159.854
C07843=1016.919,182.025,-124.811,167.547,53.008,159.856
C07844=1016.914,181.776,-124.790,167.543,53.017,159.857
C07845=1016.909,181.527,-124.768,167.538,53.028,159.858
C07846=1016.904,181.278,-124.748,167.534,53.037,159.859
C07847=1016.899,181.029,-124.726,167.530,53.047,159.860
C07848=1016.895,180.780,-124.705,167.526,53.057,159.861
C07849=1016.889,180.530,-124.684,167.522,53.067,159.862
C07850=1016.885,180.282,-124.662,167.518,53.077,159.864
C07851=1016.880,180.032,-124.641,167.514,53.086,159.865
C07852=1016.875,179.784,-124.620,167.509,53.096,159.866
C07853=1016.870,179.534,-124.599,167.505,53.106,159.867
C07854=1016.865,179.285,-124.578,167.501,53.115,159.868
C07855=1016.860,179.036,-124.556,167.498,53.125,159.869
C07856=1016.855,178.787,-124.535,167.493,53.136,159.871
C07857=1016.850,178.538,-124.515,167.489,53.145,159.872
C07858=1016.845,178.289,-124.493,167.485,53.155,159.873
C07859=1016.841,178.039,-124.472,167.481,53.165,159.874
C07860=1016.836,177.790,-124.451,167.477,53.174,159.875
C07861=1016.831,177.542,-124.429,167.473,53.185,159.876
C07862=1016.826,177.293,-124.409,167.469,53.195,159.878
C07863=1016.822,177.044,-124.388,167.465,53.204,159.879
C07864=1016.817,176.794,-124.367,167.461,53.214,159.880
C07865=1016.812,176.546,-124.346,167.457,53.224,159.881
C07866=1016.807,176.296,-124.324,167.452,53.234,159.882
C07867=1016.803,176.047,-124.303,167.449,53.244,159.883
C07868=1016.797,175.798,-124.283,167.445,53.254,159.885
C07869=1016.792,175.549,-124.261,167.441,53.263,159.886
C07870=1016.788,175.301,-124.241,167.437,53.273,159.887
C07871=1016.783,175.051,-124.220,167.434,53.283,159.888
C07872=1016.779,174.802,-124.198,167.428,53.293,159.889
C07873=1016.773,174.553,-124.178,167.425,53.303,159.891
C07874=1016.769,174.304,-124.156,167.421,53.312,159.892
C07875=1016.763,174.055,-124.135,167.417,53.322,159.893
C07876=1016.759,173.806,-124.115,167.414,53.332,159.894
C07877=1016.755,173.556,-124.093,167.409,53.341,159.895
C07878=1016.750,173.307,-124.073,167.406,53.351,159.896
C07879=1016.745,173.058,-124.052,167.401,53.362,159.898
C07880=1016.740,172.809,-124.031,167.397,53.371,159.899
C07881=1016.736,172.561,-124.010,167.393,53.381,159.900
C07882=1016.731,172.311,-123.989,167.390,53.391,159.901
C07883=1016.726,172.062,-123.968,167.386,53.400,159.902
C07884=1016.721,171.813,-123.947,167.382,53.410,159.904
C07885=1016.718,171.564,-123.926,167.378,53.420,159.905
C07886=1016.712,171.283,-123.903,167.374,53.431,159.906
C07887=1016.707,171.003,-123.879,167.370,53.442,159.907
C07888=1016.701,170.722,-123.856,167.366,53.453,159.909
C07889=1016.695,170.441,-123.832,167.360,53.465,159.910
C07890=1016.692,170.192,-123.812,167.356,53.474,159.911
C07891=1016.687,169.943,-123.790,167.353,53.484,159.912
C07892=1016.681,169.694,-123.769,167.349,53.494,159.914
C07893=1016.678,169.445,-123.748,167.345,53.503,159.915
C07894=1016.672,169.196,-123.728,167.341,53.513,159.916
C07895=1016.668,168.947,-123.707,167.338,53.524,159.917
C07896=1016.664,168.698,-123.686,167.334,53.533,159.918
C07897=1016.659,168.449,-123.665,167.330,53.543,159.920
C07898=1016.654,168.199,-123.644,167.326,53.552,159.921
C07899=1016.649,167.951,-123.624,167.323,53.562,159.922
C07900=1016.645,167.702,-123.603,167.319,53.572,159.923
C07901=1016.641,167.452,-123.583,167.315,53.582,159.924
C07902=1016.636,167.203,-123.562,167.311,53.592,159.926
C07903=1016.631,166.954,-123.541,167.307,53.601,159.927
C07904=1016.626,166.705,-123.521,167.304,53.611,159.928
C07905=1016.622,166.456,-123.500,167.300,53.621,159.929
C07906=1016.618,166.206,-123.479,167.296,53.631,159.930
C07907=1016.613,165.957,-123.458,167.293,53.641,159.932
C07908=1016.609,165.709,-123.437,167.289,53.650,159.933
C07909=1016.603,165.459,-123.417,167.285,53.660,159.934
C07910=1016.599,165.211,-123.396,167.281,53.670,159.935
C07911=1016.594,164.962,-123.375,167.278,53.680,159.936
C07912=1016.590,164.712,-123.354,167.274,53.690,159.938
C07913=1016.586,164.463,-123.334,167.270,53.699,159.939
C07914=1016.581,164.214,-123.314,167.266,53.709,159.940
C07915=1016.577,163.965,-123.293,167.262,53.719,159.941
C07916=1016.572,163.716,-123.272,167.259,53.729,159.942
C07917=1016.567,163.466,-123.251,167.255,53.739,159.944
C07918=1016.563,163.218,-123.230,167.251,53.748,159.945
C07919=1016.558,162.968,-123.211,167.249,53.758,159.946
C07920=1016.554,162.719,-123.190,167.245,53.767,159.947
C07921=1016.549,162.470,-123.169,167.241,53.778,159.948
C07922=1016.545,162.221,-123.149,167.237,53.787,159.950
C07923=1016.541,161.972,-123.127,167.234,53.797,159.951
C07924=1016.536,161.723,-123.108,167.230,53.806,159.952
C07925=1016.532,161.473,-123.087,167.226,53.817,159.953
C07926=1016.527,161.225,-123.067,167.223,53.827,159.954
C07927=1016.523,160.976,-123.045,167.219,53.836,159.956
C07928=1016.518,160.726,-123.026,167.215,53.846,159.957
C07929=1016.514,160.477,-123.005,167.212,53.855,159.958
C07930=1016.510,160.228,-122.984,167.209,53.865,159.959
C07931=1016.505,159.979,-122.963,167.205,53.875,159.960
C07932=1016.501,159.730,-122.943,167.201,53.885,159.962
C07933=1016.496,159.481,-122.923,167.197,53.894,159.963
C07934=1016.492,159.232,-122.902,167.194,53.904,159.964
C07935=1016.487,158.982,-122.882,167.190,53.914,159.965
C07936=1016.483,158.733,-122.861,167.186,53.924,159.966
C07937=1016.478,158.484,-122.840,167.184,53.933,159.968
C07938=1016.474,158.235,-122.821,167.180,53.943,159.969
C07939=1016.469,157.986,-122.800,167.177,53.953,159.970
C07940=1016.464,157.737,-122.781,167.173,53.964,159.971
C07941=1016.459,157.488,-122.760,167.169,53.973,159.973
C07942=1016.455,157.239,-122.741,167.166,53.983,159.974
C07943=1016.450,156.989,-122.721,167.162,53.993,159.975
C07944=1016.445,156.741,-122.701,167.159,54.003,159.976
C07945=1016.441,156.490,-122.680,167.155,54.014,159.978
C07946=1016.436,156.242,-122.660,167.151,54.023,159.979
C07947=1016.432,155.993,-122.641,167.148,54.033,159.980
C07948=1016.427,155.743,-122.621,167.144,54.043,159.981
C07949=1016.422,155.495,-122.601,167.141,54.053,159.983
C07950=1016.417,155.213,-122.578,167.137,54.065,159.984
C07951=1016.412,154.932,-122.556,167.133,54.076,159.986
C07952=1016.407,154.652,-122.533,167.129,54.087,159.987
C07953=1016.402,154.371,-122.511,167.125,54.098,159.988
C07954=1016.397,154.122,-122.491,167.121,54.108,159.989
C07955=1016.392,153.873,-122.471,167.118,54.118,159.991
C07956=1016.387,153.623,-122.451,167.114,54.128,159.992
C07957=1016.383,153.375,-122.431,167.110,54.138,159.993
C07958=1016.378,153.126,-122.412,167.107,54.148,159.994
C07959=1016.374,152.876,-122.392,167.103,54.158,159.996
C07960=1016.370,152.626,-122.372,167.100,54.168,159.997
C07961=1016.364,152.378,-122.352,167.096,54.178,159.998
C07962=1016.360,152.129,-122.332,167.094,54.188,159.999
C07963=1016.355,151.880,-122.313,167.090,54.198,160.001
C07964=1016.350,151.630,-122.293,167.087,54.208,160.002
C07965=1016.346,151.381,-122.274,167.083,54.218,160.003
C07966=1016.341,151.131,-122.254,167.080,54.228,160.005
C07967=1016.336,150.883,-122.234,167.076,54.238,160.006
C07968=1016.332,150.634,-122.214,167.073,54.248,160.007
C07969=1016.327,150.384,-122.194,167.069,54.258,160.008
C07970=1016.323,150.135,-122.175,167.066,54.268,160.010
C07971=1016.318,149.886,-122.155,167.062,54.278,160.011
C07972=1016.313,149.636,-122.135,167.058,54.288,160.012
C07973=1016.309,149.387,-122.116,167.055,54.298,160.013
C07974=1016.305,149.138,-122.096,167.052,54.308,160.015
C07975=1016.299,148.889,-122.076,167.048,54.318,160.016
C07976=1016.295,148.640,-122.056,167.045,54.328,160.017
C07977=1016.291,148.391,-122.037,167.042,54.338,160.019
C07978=1016.286,148.142,-122.018,167.039,54.348,160.020
C07979=1016.281,147.892,-121.998,167.035,54.358,160.021
C07980=1016.276,147.643,-121.979,167.031,54.368,160.022
C07981=1016.272,147.394,-121.959,167.028,54.378,160.024
C07982=1016.267,147.144,-121.939,167.025,54.388,160.025
C07983=1016.263,146.895,-121.920,167.021,54.399,160.026
C07984=1016.258,146.646,-121.901,167.017,54.408,160.027
C07985=1016.254,146.397,-121.881,167.014,54.418,160.029
C07986=1016.249,146.147,-121.861,167.012,54.428,160.030
C07987=1016.244,145.899,-121.842,167.008,54.438,160.031
C07988=1016.240,145.650,-121.823,167.005,54.449,160.033
C07989=1016.235,145.401,-121.803,167.001,54.458,160.034
C07990=1016.230,145.151,-121.784,166.998,54.468,160.035
C07991=1016.226,144.901,-121.765,166.994,54.479,160.036
C07992=1016.221,144.653,-121.746,166.991,54.489,160.038
C07993=1016.217,144.403,-121.726,166.988,54.499,160.039
C07994=1016.212,144.154,-121.707,166.984,54.509,160.040
C07995=1016.207,143.905,-121.688,166.981,54.519,160.041
C07996=1016.202,143.656,-121.668,166.977,54.529,160.043
C07997=1016.198,143.406,-121.650,166.975,54.539,160.044
C07998=1016.193,143.157,-121.630,166.972,54.549,160.045
C07999=1016.188,142.908,-121.611,166.968,54.560,160.047
C08000=1016.184,142.659,-121.591,166.965,54.570,160.048
C08001=1016.179,142.409,-121.573,166.962,54.580,160.049
C08002=1016.175,142.160,-121.554,166.958,54.590,160.050
C08003=1016.170,141.911,-121.534,166.954,54.600,160.052
C08004=1016.165,141.662,-121.515,166.951,54.610,160.053
C08005=1016.161,141.413,-121.496,166.948,54.620,160.054
C08006=1016.156,141.163,-121.477,166.946,54.630,160.056
C08007=1016.151,140.914,-121.458,166.942,54.640,160.057
C08008=1016.146,140.665,-121.438,166.938,54.650,160.058
C08009=1016.142,140.415,-121.419,166.935,54.660,160.060
C08010=1016.137,140.166,-121.400,166.932,54.671,160.061
C08011=1016.133,139.917,-121.381,166.928,54.681,160.062
C08012=1016.129,139.668,-121.361,166.925,54.690,160.063
C08013=1016.124,139.419,-121.343,166.922,54.700,160.065
C08014=1016.119,139.138,-121.321,166.919,54.712,160.066
C08015=1016.114,138.857,-121.299,166.915,54.723,160.068
C08016=1016.108,138.576,-121.279,166.911,54.734,160.069
C08017=1016.103,138.295,-121.257,166.907,54.746,160.071
C08018=1016.099,138.046,-121.237,166.905,54.756,160.072
C08019=1016.094,137.797,-121.219,166.902,54.766,160.073
C08020=1016.089,137.547,-121.199,166.898,54.776,160.075
C08021=1016.084,137.298,-121.181,166.895,54.787,160.076
C08022=1016.080,137.048,-121.162,166.891,54.796,160.077
C08023=1016.075,136.800,-121.143,166.888,54.807,160.078
C08024=1016.071,136.550,-121.124,166.885,54.817,160.080
C08025=1016.066,136.301,-121.105,166.882,54.827,160.081
C08026=1016.062,136.052,-121.086,166.879,54.837,160.083
C08027=1016.057,135.803,-121.068,166.876,54.847,160.084
C08028=1016.053,135.553,-121.049,166.872,54.857,160.085
C08029=1016.047,135.305,-121.030,166.869,54.867,160.086
C08030=1016.043,135.054,-121.011,166.866,54.878,160.088
C08031=1016.038,134.805,-120.992,166.862,54.888,160.089
C08032=1016.033,134.556,-120.974,166.860,54.898,160.090
C08033=1016.029,134.306,-120.955,166.857,54.908,160.092
C08034=1016.024,134.058,-120.936,166.854,54.918,160.093
C08035=1016.020,133.808,-120.917,166.850,54.928,160.094
C08036=1016.015,133.559,-120.899,166.847,54.938,160.095
C08037=1016.010,133.310,-120.880,166.843,54.949,160.097
C08038=1016.006,133.060,-120.862,166.840,54.959,160.098
C08039=1016.001,132.812,-120.843,166.838,54.969,160.100
C08040=1015.997,132.562,-120.824,166.835,54.979,160.101
C08041=1015.992,132.313,-120.805,166.831,54.989,160.102
C08042=1015.987,132.064,-120.787,166.828,54.999,160.103
C08043=1015.983,131.814,-120.768,166.825,55.010,160.105
C08044=1015.978,131.565,-120.749,166.822,55.019,160.106
C08045=1015.973,131.316,-120.731,166.819,55.030,160.108
C08046=1015.969,131.066,-120.712,166.815,55.039,160.109
C08047=1015.964,130.818,-120.694,166.812,55.050,160.110
C08048=1015.960,130.568,-120.675,166.809,55.060,160.111
C08049=1015.955,130.319,-120.657,166.807,55.070,160.113
C08050=1015.950,130.070,-120.638,166.804,55.080,160.114
C08051=1015.946,129.820,-120.619,166.800,55.090,160.115
C08052=1015.941,129.571,-120.601,166.797,55.100,160.117
C08053=1015.936,129.322,-120.583,166.794,55.111,160.118
C08054=1015.931,129.073,-120.564,166.791,55.121,160.119
C08055=1015.927,128.823,-120.545,166.788,55.131,160.121
C08056=1015.922,128.574,-120.527,166.785,55.141,160.122
C08057=1015.918,128.325,-120.509,166.782,55.152,160.123
C08058=1015.913,128.075,-120.491,166.779,55.162,160.125
C08059=1015.908,127.826,-120.472,166.775,55.173,160.126
C08060=1015.903,127.576,-120.454,166.772,55.183,160.127
C08061=1015.899,127.327,-120.436,166.769,55.193,160.129
C08062=1015.894,127.078,-120.418,166.766,55.204,160.130
C08063=1015.889,126.828,-120.400,166.764,55.214,160.132
C08064=1015.884,126.579,-120.382,166.761,55.224,160.133
C08065=1015.879,126.330,-120.363,166.757,55.234,160.134
C08066=1015.874,126.081,-120.345,166.754,55.244,160.135
C08067=1015.870,125.832,-120.326,166.751,55.254,160.137
C08068=1015.865,125.582,-120.308,166.748,55.265,160.138
C08069=1015.860,125.333,-120.290,166.744,55.275,160.139
C08070=1015.855,125.084,-120.272,166.742,55.285,160.141
C08071=1015.850,124.834,-120.254,166.739,55.295,160.142
C08072=1015.846,124.585,-120.236,166.736,55.306,160.144
C08073=1015.841,124.336,-120.218,166.733,55.316,160.145
C08074=1015.837,124.087,-120.200,166.730,55.327,160.146
C08075=1015.832,123.838,-120.181,166.726,55.336,160.147
C08076=1015.827,123.588,-120.163,166.724,55.346,160.149
C08077=1015.822,123.339,-120.145,166.721,55.357,160.150
C08078=1015.817,123.058,-120.124,166.717,55.368,160.152
C08079=1015.812,122.777,-120.105,166.713,55.380,160.153
C08080=1015.807,122.495,-120.084,166.710,55.391,160.155
C08081=1015.801,122.214,-120.064,166.708,55.403,160.157
C08082=1015.797,121.965,-120.046,166.704,55.413,160.158
C08083=1015.792,121.716,-120.028,166.701,55.423,160.159
C08084=1015.788,121.467,-120.010,166.698,55.434,160.160
C08085=1015.783,121.217,-119.991,166.696,55.444,160.162
C08086=1015.778,120.968,-119.973,166.693,55.454,160.163
C08087=1015.773,120.719,-119.955,166.689,55.464,160.164
C08088=1015.768,120.469,-119.937,166.686,55.474,160.166
C08089=1015.764,120.221,-119.919,166.684,55.484,160.167
C08090=1015.759,119.971,-119.901,166.681,55.495,160.169
C08091=1015.755,119.721,-119.884,166.678,55.505,160.170
C08092=1015.750,119.472,-119.865,166.674,55.515,160.171
C08093=1015.745,119.223,-119.847,166.672,55.525,160.173
C08094=1015.741,118.973,-119.829,166.669,55.535,160.174
C08095=1015.736,118.725,-119.811,166.666,55.546,160.175
C08096=1015.732,118.475,-119.793,166.663,55.556,160.177
C08097=1015.727,118.226,-119.775,166.660,55.565,160.178
C08098=1015.722,117.976,-119.757,166.657,55.576,160.179
C08099=1015.718,117.726,-119.739,166.654,55.586,160.181
C08100=1015.714,117.478,-119.721,166.651,55.596,160.182
C08101=1015.709,117.228,-119.703,166.648,55.606,160.183
C08102=1015.705,116.979,-119.685,166.645,55.616,160.185
C08103=1015.700,116.730,-119.666,166.643,55.626,160.186
C08104=1015.696,116.480,-119.649,166.640,55.636,160.187
C08105=1015.691,116.231,-119.631,166.637,55.647,160.189
C08106=1015.686,115.982,-119.613,166.634,55.657,160.190
C08107=1015.682,115.732,-119.595,166.631,55.666,160.191
C08108=1015.677,115.484,-119.577,166.628,55.677,160.193
C08109=1015.673,115.234,-119.560,166.625,55.687,160.194
C08110=1015.668,114.984,-119.541,166.622,55.697,160.195
C08111=1015.663,114.735,-119.523,166.619,55.707,160.197
C08112=1015.659,114.486,-119.505,166.617,55.717,160.198
C08113=1015.655,114.236,-119.488,166.614,55.727,160.199
C08114=1015.650,113.987,-119.470,166.611,55.737,160.201
C08115=1015.645,113.738,-119.452,166.609,55.747,160.202
C08116=1015.641,113.489,-119.434,166.605,55.757,160.203
C08117=1015.637,113.239,-119.416,166.602,55.768,160.205
C08118=1015.632,112.990,-119.398,166.600,55.778,160.206
C08119=1015.628,112.741,-119.381,166.597,55.787,160.207
C08120=1015.623,112.492,-119.362,166.595,55.797,160.209
C08121=1015.618,112.242,-119.345,166.591,55.807,160.210
C08122=1015.614,111.992,-119.327,166.588,55.818,160.211
C08123=1015.609,111.744,-119.309,166.586,55.828,160.213
C08124=1015.604,111.494,-119.292,166.583,55.838,160.214
C08125=1015.599,111.245,-119.274,166.580,55.848,160.215
C08126=1015.596,110.995,-119.257,166.577,55.859,160.217
C08127=1015.590,110.746,-119.239,166.575,55.869,160.218
C08128=1015.586,110.496,-119.222,166.572,55.879,160.219
C08129=1015.581,110.247,-119.204,166.568,55.889,160.221
C08130=1015.577,109.998,-119.187,166.566,55.899,160.222
C08131=1015.571,109.749,-119.169,166.563,55.909,160.224
C08132=1015.567,109.499,-119.152,166.560,55.920,160.225
C08133=1015.563,109.250,-119.134,166.558,55.929,160.226
C08134=1015.557,109.001,-119.117,166.555,55.940,160.228
C08135=1015.553,108.751,-119.099,166.552,55.950,160.229
C08136=1015.548,108.502,-119.082,166.549,55.961,160.230
C08137=1015.544,108.252,-119.065,166.547,55.971,160.232
C08138=1015.539,108.003,-119.047,166.543,55.981,160.233
C08139=1015.534,107.754,-119.030,166.540,55.991,160.234
C08140=1015.530,107.504,-119.013,166.537,56.002,160.236
C08141=1015.524,107.255,-118.995,166.535,56.012,160.237
C08142=1015.517,106.847,-118.967,166.531,56.029,160.239
C08143=1015.509,106.439,-118.939,166.526,56.046,160.242
C08144=1015.502,106.030,-118.911,166.522,56.062,160.244
C08145=1015.494,105.622,-118.883,166.517,56.079,160.246
C08146=1015.487,105.250,-118.856,166.513,56.094,160.248
C08147=1015.480,104.879,-118.831,166.508,56.109,160.250
C08148=1015.473,104.508,-118.806,166.505,56.124,160.252
C08149=1015.467,104.137,-118.780,166.500,56.140,160.254
C08150=1015.461,103.887,-118.762,166.498,56.149,160.256
C08151=1015.457,103.637,-118.745,166.495,56.160,160.257
C08152=1015.452,103.389,-118.728,166.493,56.170,160.259
C08153=1015.447,103.139,-118.711,166.489,56.180,160.260
C08154=1015.443,102.890,-118.694,166.487,56.190,160.261
C08155=1015.438,102.640,-118.676,166.485,56.200,160.263
C08156=1015.433,102.391,-118.660,166.481,56.210,160.264
C08157=1015.429,102.141,-118.642,166.478,56.221,160.265
C08158=1015.424,101.893,-118.625,166.476,56.231,160.267
C08159=1015.420,101.643,-118.608,166.473,56.241,160.268
C08160=1015.414,101.393,-118.591,166.470,56.251,160.269
C08161=1015.411,101.144,-118.574,166.468,56.261,160.271
C08162=1015.405,100.894,-118.557,166.465,56.271,160.272
C08163=1015.401,100.646,-118.539,166.463,56.281,160.273
C08164=1015.396,100.396,-118.522,166.460,56.291,160.275
C08165=1015.392,100.147,-118.505,166.457,56.302,160.276
C08166=1015.388,99.897,-118.488,166.455,56.312,160.278
C08167=1015.383,99.648,-118.471,166.451,56.322,160.279
C08168=1015.378,99.399,-118.453,166.450,56.332,160.280
C08169=1015.374,99.150,-118.437,166.446,56.342,160.281
C08170=1015.369,98.900,-118.419,166.444,56.352,160.283
C08171=1015.364,98.651,-118.403,166.441,56.363,160.284
C08172=1015.359,98.401,-118.386,166.438,56.372,160.285
C08173=1015.355,98.152,-118.369,166.435,56.383,160.287
C08174=1015.350,97.902,-118.352,166.433,56.393,160.288
C08175=1015.346,97.653,-118.336,166.430,56.403,160.290
C08176=1015.340,97.403,-118.319,166.427,56.414,160.291
C08177=1015.336,97.155,-118.302,166.425,56.424,160.293
C08178=1015.331,96.905,-118.285,166.422,56.434,160.294
C08179=1015.327,96.656,-118.268,166.419,56.444,160.295
C08180=1015.321,96.406,-118.251,166.417,56.454,160.297
C08181=1015.317,96.157,-118.235,166.414,56.465,160.298
C08182=1015.312,95.907,-118.219,166.412,56.474,160.299
C08183=1015.307,95.658,-118.202,166.409,56.485,160.301
C08184=1015.303,95.408,-118.185,166.406,56.496,160.302
C08185=1015.298,95.159,-118.168,166.404,56.505,160.303
C08186=1015.293,94.909,-118.152,166.401,56.516,160.305
C08187=1015.288,94.660,-118.135,166.398,56.525,160.306
C08188=1015.284,94.410,-118.118,166.396,56.536,160.308
C08189=1015.279,94.161,-118.101,166.393,56.546,160.309
C08190=1015.275,93.912,-118.085,166.391,56.556,160.310
C08191=1015.270,93.663,-118.068,166.388,56.566,160.312
C08192=1015.265,93.414,-118.051,166.385,56.576,160.313
C08193=1015.261,93.163,-118.035,166.383,56.586,160.314
C08194=1015.256,92.914,-118.018,166.380,56.597,160.316
C08195=1015.251,92.664,-118.001,166.378,56.606,160.317
C08196=1015.246,92.416,-117.985,166.375,56.617,160.319
C08197=1015.242,92.167,-117.968,166.372,56.627,160.320
C08198=1015.237,91.917,-117.951,166.370,56.637,160.321
C08199=1015.233,91.668,-117.934,166.366,56.647,160.322
C08200=1015.227,91.418,-117.917,166.365,56.657,160.324
C08201=1015.223,91.168,-117.902,166.361,56.667,160.325
C08202=1015.218,90.888,-117.883,166.359,56.678,160.327
C08203=1015.212,90.607,-117.864,166.356,56.690,160.328
C08204=1015.208,90.327,-117.845,166.353,56.701,160.330
C08205=1015.202,90.046,-117.826,166.350,56.713,160.331
C08206=1015.198,89.797,-117.810,166.348,56.723,160.333
C08207=1015.193,89.547,-117.794,166.345,56.733,160.334
C08208=1015.189,89.297,-117.777,166.342,56.742,160.335
C08209=1015.184,89.048,-117.760,166.340,56.753,160.337
C08210=1015.179,88.799,-117.743,166.337,56.762,160.338
C08211=1015.175,88.549,-117.727,166.335,56.773,160.340
C08212=1015.170,88.300,-117.711,166.332,56.784,160.341
C08213=1015.165,88.051,-117.694,166.330,56.793,160.342
C08214=1015.161,87.801,-117.678,166.327,56.804,160.344
C08215=1015.156,87.551,-117.661,166.325,56.813,160.345
C08216=1015.150,87.302,-117.646,166.322,56.824,160.346
C08217=1015.145,87.052,-117.629,166.319,56.835,160.348
C08218=1015.141,86.803,-117.613,166.317,56.844,160.349
C08219=1015.136,86.554,-117.597,166.314,56.855,160.351
C08220=1015.131,86.304,-117.580,166.311,56.865,160.352
C08221=1015.127,86.055,-117.565,166.309,56.875,160.353
C08222=1015.122,85.806,-117.548,166.306,56.885,160.355
C08223=1015.118,85.556,-117.532,166.304,56.895,160.356
C08224=1015.113,85.306,-117.515,166.301,56.906,160.358
C08225=1015.108,85.058,-117.499,166.299,56.915,160.359
C08226=1015.103,84.808,-117.484,166.296,56.926,160.360
C08227=1015.098,84.559,-117.467,166.293,56.936,160.362
C08228=1015.094,84.309,-117.451,166.291,56.946,160.363
C08229=1015.089,84.060,-117.435,166.288,56.956,160.364
C08230=1015.084,83.810,-117.419,166.287,56.966,160.366
C08231=1015.079,83.561,-117.402,166.283,56.976,160.367
C08232=1015.075,83.311,-117.386,166.282,56.986,160.369
C08233=1015.070,83.062,-117.369,166.278,56.996,160.370
C08234=1015.066,82.812,-117.354,166.276,57.006,160.371
C08235=1015.060,82.563,-117.338,166.273,57.017,160.373
C08236=1015.056,82.314,-117.322,166.271,57.026,160.374
C08237=1015.051,82.064,-117.305,166.269,57.037,160.375
C08238=1015.046,81.815,-117.289,166.266,57.046,160.377
C08239=1015.042,81.566,-117.273,166.264,57.057,160.378
C08240=1015.037,81.316,-117.257,166.260,57.067,160.379
C08241=1015.032,81.066,-117.240,166.258,57.077,160.381
C08242=1015.028,80.817,-117.225,166.257,57.087,160.382
C08243=1015.023,80.567,-117.209,166.253,57.097,160.383
C08244=1015.018,80.319,-117.193,166.251,57.106,160.385
C08245=1015.013,80.068,-117.177,166.248,57.117,160.386
C08246=1015.009,79.819,-117.160,166.246,57.127,160.388
C08247=1015.004,79.570,-117.144,166.243,57.136,160.389
C08248=1015.000,79.321,-117.128,166.241,57.147,160.390
C08249=1014.995,79.070,-117.112,166.238,57.157,160.391
C08250=1014.991,78.821,-117.096,166.236,57.166,160.393
C08251=1014.986,78.572,-117.080,166.233,57.177,160.394
C08252=1014.981,78.323,-117.064,166.231,57.187,160.396
C08253=1014.976,78.074,-117.048,166.228,57.197,160.397
C08254=1014.971,77.823,-117.032,166.226,57.207,160.398
C08255=1014.967,77.574,-117.016,166.224,57.216,160.400
C08256=1014.963,77.325,-117.000,166.221,57.226,160.401
C08257=1014.958,77.075,-116.984,166.219,57.236,160.402
C08258=1014.954,76.826,-116.968,166.216,57.247,160.404
C08259=1014.948,76.576,-116.952,166.214,57.256,160.405
C08260=1014.944,76.327,-116.936,166.211,57.266,160.406
C08261=1014.939,76.077,-116.920,166.209,57.276,160.408
C08262=1014.934,75.828,-116.905,166.206,57.286,160.409
C08263=1014.930,75.579,-116.889,166.204,57.296,160.410
C08264=1014.925,75.329,-116.873,166.201,57.307,160.412
C08265=1014.920,75.079,-116.857,166.199,57.316,160.413
C08266=1014.915,74.799,-116.840,166.197,57.328,160.415
C08267=1014.910,74.519,-116.821,166.193,57.339,160.416
C08268=1014.904,74.238,-116.804,166.191,57.350,160.418
C08269=1014.899,73.957,-116.786,166.188,57.362,160.419
C08270=1014.894,73.708,-116.771,166.186,57.371,160.421
C08271=1014.890,73.459,-116.756,166.183,57.382,160.422
C08272=1014.885,73.210,-116.739,166.181,57.391,160.423
C08273=1014.879,72.960,-116.724,166.178,57.401,160.425
C08274=1014.875,72.710,-116.708,166.176,57.412,160.426
C08275=1014.870,72.461,-116.693,166.174,57.421,160.428
C08276=1014.866,72.211,-116.677,166.171,57.431,160.429
C08277=1014.861,71.962,-116.661,166.169,57.441,160.430
C08278=1014.856,71.712,-116.646,166.166,57.452,160.432
C08279=1014.852,71.463,-116.630,166.164,57.461,160.433
C08280=1014.847,71.214,-116.615,166.161,57.471,160.434
C08281=1014.842,70.964,-116.598,166.159,57.481,160.435
C08282=1014.837,70.715,-116.583,166.157,57.491,160.437
C08283=1014.832,70.465,-116.567,166.154,57.501,160.438
C08284=1014.828,70.215,-116.551,166.152,57.511,160.440
C08285=1014.823,69.966,-116.536,166.149,57.521,160.441
C08286=1014.819,69.717,-116.520,166.147,57.531,160.442
C08287=1014.814,69.467,-116.505,166.144,57.541,160.443
C08288=1014.809,69.218,-116.489,166.142,57.551,160.445
C08289=1014.804,68.969,-116.474,166.140,57.560,160.446
C08290=1014.800,68.719,-116.459,166.137,57.571,160.448
C08291=1014.795,68.470,-116.443,166.135,57.580,160.449
C08292=1014.791,68.220,-116.428,166.133,57.590,160.450
C08293=1014.785,67.970,-116.412,166.130,57.600,160.451
C08294=1014.781,67.721,-116.396,166.128,57.610,160.453
C08295=1014.776,67.471,-116.381,166.125,57.620,160.454
C08296=1014.771,67.222,-116.365,166.123,57.630,160.456
C08297=1014.766,66.972,-116.350,166.121,57.639,160.457
C08298=1014.761,66.723,-116.335,166.118,57.649,160.458
C08299=1014.757,66.474,-116.319,166.116,57.659,160.460
C08300=1014.752,66.224,-116.305,166.113,57.670,160.461
C08301=1014.748,65.974,-116.289,166.111,57.679,160.462
C08302=1014.743,65.725,-116.274,166.109,57.689,160.464
C08303=1014.738,65.476,-116.259,166.106,57.699,160.465
C08304=1014.734,65.226,-116.243,166.104,57.709,160.466
C08305=1014.729,64.977,-116.228,166.101,57.719,160.468
C08306=1014.724,64.727,-116.212,166.099,57.728,160.469
C08307=1014.720,64.477,-116.197,166.097,57.739,160.471
C08308=1014.715,64.228,-116.182,166.094,57.749,160.472
C08309=1014.710,63.978,-116.167,166.092,57.759,160.473
C08310=1014.705,63.729,-116.151,166.090,57.768,160.475
C08311=1014.700,63.480,-116.136,166.087,57.778,160.476
C08312=1014.696,63.230,-116.120,166.085,57.788,160.477
C08313=1014.691,62.980,-116.106,166.082,57.798,160.478
C08314=1014.686,62.731,-116.091,166.080,57.808,160.480
C08315=1014.682,62.482,-116.075,166.078,57.817,160.481
C08316=1014.677,62.232,-116.061,166.075,57.827,160.482
C08317=1014.672,61.982,-116.045,166.074,57.838,160.484
C08318=1014.667,61.733,-116.030,166.071,57.848,160.485
C08319=1014.662,61.483,-116.016,166.069,57.857,160.487
C08320=1014.657,61.234,-116.001,166.065,57.868,160.488
C08321=1014.652,60.984,-115.986,166.063,57.877,160.489
C08322=1014.647,60.735,-115.971,166.062,57.888,160.491
C08323=1014.642,60.486,-115.956,166.059,57.898,160.492
C08324=1014.638,60.236,-115.941,166.057,57.907,160.493
C08325=1014.633,59.986,-115.926,166.054,57.917,160.495
C08326=1014.628,59.737,-115.912,166.052,57.927,160.496
C08327=1014.623,59.487,-115.896,166.049,57.937,160.497
C08328=1014.618,59.237,-115.882,166.047,57.947,160.499
C08329=1014.613,58.988,-115.867,166.045,57.956,160.500
C08330=1014.607,58.708,-115.850,166.042,57.968,160.502
C08331=1014.602,58.427,-115.834,166.040,57.979,160.503
C08332=1014.596,58.147,-115.817,166.037,57.990,160.505
C08333=1014.591,57.866,-115.800,166.034,58.001,160.506
C08334=1014.586,57.617,-115.785,166.032,58.011,160.507
C08335=1014.581,57.367,-115.770,166.030,58.021,160.509
C08336=1014.577,57.118,-115.756,166.027,58.031,160.510
C08337=1014.572,56.869,-115.741,166.025,58.041,160.511
C08338=1014.567,56.619,-115.726,166.023,58.050,160.513
C08339=1014.562,56.370,-115.711,166.020,58.060,160.514
C08340=1014.558,56.120,-115.697,166.018,58.070,160.515
C08341=1014.553,55.871,-115.681,166.016,58.080,160.517
C08342=1014.548,55.621,-115.667,166.013,58.090,160.518
C08343=1014.543,55.371,-115.653,166.011,58.099,160.519
C08344=1014.538,55.122,-115.637,166.009,58.109,160.521
C08345=1014.534,54.872,-115.623,166.006,58.119,160.522
C08346=1014.529,54.623,-115.608,166.004,58.129,160.523
C08347=1014.524,54.373,-115.594,166.002,58.139,160.525
C08348=1014.519,54.124,-115.578,166.000,58.148,160.526
C08349=1014.514,53.874,-115.564,165.997,58.158,160.527
C08350=1014.509,53.625,-115.549,165.995,58.168,160.529
C08351=1014.505,53.375,-115.534,165.993,58.177,160.530
C08352=1014.500,53.126,-115.520,165.990,58.187,160.531
C08353=1014.495,52.877,-115.505,165.988,58.197,160.532
C08354=1014.491,52.627,-115.491,165.986,58.207,160.534
C08355=1014.486,52.377,-115.475,165.984,58.216,160.535
C08356=1014.481,52.127,-115.461,165.980,58.226,160.536
C08357=1014.476,51.878,-115.446,165.979,58.235,160.538
C08358=1014.472,51.629,-115.432,165.977,58.245,160.539
C08359=1014.467,51.379,-115.417,165.975,58.255,160.540
C08360=1014.462,51.130,-115.402,165.973,58.265,160.542
C08361=1014.457,50.880,-115.388,165.969,58.274,160.543
C08362=1014.452,50.631,-115.372,165.967,58.284,160.544
C08363=1014.447,50.381,-115.358,165.965,58.293,160.546
C08364=1014.443,50.132,-115.344,165.963,58.302,160.547
C08365=1014.438,49.882,-115.329,165.961,58.312,160.548
C08366=1014.434,49.633,-115.314,165.959,58.322,160.550
C08367=1014.429,49.383,-115.300,165.956,58.332,160.551
C08368=1014.424,49.133,-115.285,165.954,58.341,160.552
C08369=1014.420,48.884,-115.271,165.952,58.351,160.553
C08370=1014.415,48.634,-115.256,165.950,58.360,160.555
C08371=1014.410,48.385,-115.241,165.947,58.369,160.556
C08372=1014.405,48.135,-115.226,165.946,58.379,160.557
C08373=1014.401,47.886,-115.212,165.942,58.389,160.558
C08374=1014.396,47.637,-115.197,165.940,58.398,160.560
C08375=1014.391,47.387,-115.183,165.938,58.408,160.561
C08376=1014.386,47.137,-115.168,165.936,58.417,160.562
C08377=1014.382,46.888,-115.153,165.934,58.427,160.563
C08378=1014.377,46.638,-115.139,165.931,58.436,160.565
C08379=1014.373,46.389,-115.125,165.930,58.445,160.566
C08380=1014.367,46.139,-115.109,165.927,58.454,160.567
C08381=1014.364,45.890,-115.095,165.925,58.464,160.569
C08382=1014.359,45.640,-115.080,165.923,58.473,160.570
C08383=1014.355,45.390,-115.066,165.921,58.483,160.571
C08384=1014.350,45.141,-115.051,165.918,58.492,160.572
C08385=1014.345,44.892,-115.037,165.916,58.502,160.573
C08386=1014.341,44.642,-115.022,165.913,58.511,160.575
C08387=1014.336,44.392,-115.008,165.911,58.521,160.576
C08388=1014.331,44.143,-114.992,165.909,58.530,160.577
C08389=1014.327,43.893,-114.978,165.907,58.540,160.578
C08390=1014.322,43.643,-114.964,165.905,58.549,160.580
C08391=1014.317,43.394,-114.949,165.902,58.558,160.581
C08392=1014.313,43.145,-114.935,165.900,58.567,160.582
C08393=1014.308,42.895,-114.920,165.898,58.576,160.583
C08394=1014.303,42.614,-114.904,165.896,58.586,160.585
C08395=1014.297,42.334,-114.888,165.894,58.597,160.586
C08396=1014.292,42.054,-114.871,165.891,58.607,160.587
C08397=1014.287,41.773,-114.855,165.889,58.618,160.589
C08398=1014.282,41.523,-114.841,165.886,58.627,160.590
C08399=1014.277,41.275,-114.827,165.884,58.637,160.592
C08400=1014.272,41.025,-114.813,165.882,58.646,160.593
C08401=1014.268,40.775,-114.798,165.880,58.656,160.594
C08402=1014.264,40.526,-114.784,165.877,58.665,160.595
C08403=1014.258,40.276,-114.771,165.875,58.675,160.597
C08404=1014.253,40.026,-114.756,165.872,58.684,160.598
C08405=1014.249,39.777,-114.742,165.870,58.693,160.599
C08406=1014.244,39.527,-114.728,165.868,58.703,160.600
C08407=1014.239,39.277,-114.714,165.866,58.712,160.601
C08408=1014.235,39.028,-114.700,165.864,58.722,160.603
C08409=1014.229,38.779,-114.686,165.862,58.731,160.604
C08410=1014.225,38.530,-114.672,165.859,58.740,160.605
C08411=1014.221,38.280,-114.657,165.857,58.749,160.606
C08412=1014.216,38.030,-114.643,165.855,58.758,160.608
C08413=1014.211,37.781,-114.629,165.853,58.767,160.609
C08414=1014.206,37.531,-114.615,165.851,58.777,160.610
C08415=1014.201,37.281,-114.600,165.848,58.786,160.611
C08416=1014.197,37.032,-114.587,165.846,58.795,160.612
C08417=1014.192,36.782,-114.573,165.844,58.805,160.614
C08418=1014.188,36.533,-114.559,165.842,58.814,160.615
C08419=1014.183,36.283,-114.544,165.839,58.823,160.616
C08420=1014.178,36.033,-114.531,165.837,58.832,160.617
C08421=1014.174,35.784,-114.517,165.835,58.842,160.619
C08422=1014.168,35.534,-114.503,165.833,58.851,160.620
C08423=1014.164,35.285,-114.490,165.831,58.861,160.621
C08424=1014.159,35.035,-114.475,165.829,58.870,160.622
C08425=1014.153,34.785,-114.462,165.826,58.879,160.624
C08426=1014.149,34.536,-114.447,165.825,58.889,160.625
C08427=1014.144,34.286,-114.434,165.822,58.898,160.626
C08428=1014.140,34.037,-114.420,165.820,58.907,160.627
C08429=1014.134,33.787,-114.406,165.818,58.916,160.628
C08430=1014.130,33.538,-114.392,165.816,58.926,160.630
C08431=1014.125,33.288,-114.379,165.813,58.935,160.631
C08432=1014.120,33.038,-114.365,165.811,58.944,160.632
C08433=1014.116,32.789,-114.351,165.809,58.953,160.633
C08434=1014.110,32.539,-114.338,165.807,58.963,160.635
C08435=1014.106,32.290,-114.324,165.805,58.972,160.636
C08436=1014.101,32.040,-114.310,165.802,58.981,160.637
C08437=1014.097,31.791,-114.296,165.800,58.990,160.638
C08438=1014.091,31.541,-114.283,165.798,58.999,160.639
C08439=1014.087,31.292,-114.269,165.796,59.009,160.641
C08440=1014.082,31.042,-114.255,165.795,59.017,160.642
C08441=1014.078,30.792,-114.241,165.792,59.026,160.643
C08442=1014.073,30.543,-114.228,165.790,59.036,160.644
C08443=1014.068,30.294,-114.214,165.787,59.045,160.646
C08444=1014.063,30.043,-114.200,165.785,59.054,160.647
C08445=1014.058,29.794,-114.187,165.783,59.063,160.648
C08446=1014.054,29.545,-114.172,165.780,59.072,160.649
C08447=1014.049,29.295,-114.160,165.778,59.081,160.650
C08448=1014.044,29.045,-114.145,165.776,59.090,160.651
C08449=1014.039,28.796,-114.132,165.775,59.099,160.653
C08450=1014.035,28.546,-114.118,165.772,59.108,160.654
C08451=1014.030,28.297,-114.104,165.770,59.117,160.655
C08452=1014.025,28.047,-114.091,165.768,59.126,160.656
C08453=1014.021,27.797,-114.077,165.765,59.135,160.657
C08454=1014.015,27.548,-114.063,165.763,59.144,160.658
C08455=1014.012,27.298,-114.050,165.762,59.153,160.660
C08456=1014.006,27.049,-114.036,165.759,59.162,160.661
C08457=1014.001,26.799,-114.023,165.757,59.171,160.662
C08458=1013.996,26.519,-114.008,165.754,59.181,160.663
C08459=1013.990,26.238,-113.993,165.752,59.191,160.664
C08460=1013.985,25.958,-113.977,165.750,59.201,160.666
C08461=1013.980,25.678,-113.962,165.747,59.212,160.667
C08462=1013.975,25.428,-113.949,165.745,59.221,160.668
C08463=1013.970,25.179,-113.935,165.743,59.230,160.670
C08464=1013.965,24.929,-113.922,165.741,59.238,160.671
C08465=1013.961,24.679,-113.909,165.739,59.247,160.672
C08466=1013.957,24.430,-113.895,165.737,59.257,160.673
C08467=1013.951,24.180,-113.882,165.734,59.266,160.674
C08468=1013.947,23.931,-113.869,165.732,59.275,160.676
C08469=1013.941,23.681,-113.855,165.730,59.284,160.677
C08470=1013.937,23.431,-113.843,165.729,59.293,160.678
C08471=1013.933,23.182,-113.828,165.726,59.302,160.679
C08472=1013.927,22.932,-113.815,165.724,59.311,160.680
C08473=1013.923,22.683,-113.802,165.721,59.319,160.681
C08474=1013.917,22.433,-113.789,165.719,59.328,160.682
C08475=1013.913,22.183,-113.776,165.718,59.337,160.684
C08476=1013.909,21.934,-113.762,165.715,59.346,160.685
C08477=1013.904,21.684,-113.749,165.713,59.355,160.686
C08478=1013.899,21.435,-113.736,165.710,59.364,160.687
C08479=1013.894,21.185,-113.722,165.709,59.372,160.688
C08480=1013.889,20.935,-113.709,165.707,59.381,160.689
C08481=1013.884,20.686,-113.696,165.704,59.390,160.691
C08482=1013.880,20.436,-113.682,165.703,59.398,160.692
C08483=1013.875,20.187,-113.669,165.700,59.407,160.693
C08484=1013.871,19.937,-113.656,165.698,59.417,160.694
C08485=1013.865,19.688,-113.643,165.696,59.426,160.695
C08486=1013.860,19.438,-113.630,165.694,59.434,160.696
C08487=1013.857,19.188,-113.616,165.692,59.443,160.697
C08488=1013.851,18.938,-113.603,165.689,59.452,160.698
C08489=1013.847,18.689,-113.590,165.688,59.460,160.699
C08490=1013.841,18.439,-113.577,165.685,59.469,160.701
C08491=1013.837,18.189,-113.564,165.683,59.478,160.702
C08492=1013.832,17.940,-113.551,165.681,59.486,160.703
C08493=1013.827,17.691,-113.538,165.679,59.495,160.704
C08494=1013.822,17.441,-113.524,165.677,59.504,160.705
C08495=1013.818,17.191,-113.512,165.675,59.512,160.706
C08496=1013.813,16.942,-113.499,165.673,59.521,160.707
C08497=1013.808,16.692,-113.486,165.671,59.531,160.709
C08498=1013.803,16.442,-113.473,165.669,59.538,160.710
C08499=1013.798,16.193,-113.459,165.666,59.548,160.711
C08500=1013.793,15.943,-113.446,165.664,59.556,160.712
C08501=1013.789,15.694,-113.433,165.662,59.565,160.713
C08502=1013.785,15.444,-113.420,165.660,59.573,160.714
C08503=1013.780,15.194,-113.407,165.657,59.582,160.715
C08504=1013.775,14.944,-113.394,165.656,59.590,160.716
C08505=1013.771,14.695,-113.381,165.653,59.599,160.717
C08506=1013.766,14.445,-113.369,165.651,59.607,160.718
C08507=1013.761,14.196,-113.355,165.649,59.616,160.719
C08508=1013.756,13.946,-113.342,165.646,59.625,160.720
C08509=1013.751,13.697,-113.329,165.645,59.634,160.722
C08510=1013.747,13.447,-113.316,165.642,59.642,160.722
C08511=1013.742,13.197,-113.303,165.641,59.651,160.724
C08512=1013.737,12.947,-113.290,165.638,59.659,160.725
C08513=1013.733,12.698,-113.278,165.637,59.668,160.726
C08514=1013.727,12.448,-113.265,165.634,59.676,160.727
C08515=1013.722,12.199,-113.252,165.632,59.685,160.728
C08516=1013.717,11.949,-113.240,165.630,59.693,160.729
C08517=1013.713,11.699,-113.227,165.628,59.702,160.730
C08518=1013.708,11.450,-113.215,165.625,59.711,160.731
C08519=1013.703,11.200,-113.202,165.624,59.720,160.733
C08520=1013.698,10.950,-113.189,165.621,59.728,160.733
C08521=1013.694,10.701,-113.177,165.620,59.737,160.735
C08522=1013.688,10.422,-113.163,165.617,59.746,160.736
C08523=1013.682,10.143,-113.149,165.615,59.755,160.737
C08524=1013.677,9.864,-113.135,165.613,59.765,160.739
C08525=1013.672,9.586,-113.121,165.610,59.775,160.739
C08526=1013.667,9.336,-113.108,165.608,59.783,160.741
C08527=1013.662,9.086,-113.095,165.605,59.791,160.741
C08528=1013.657,8.837,-113.083,165.604,59.800,160.743
C08529=1013.652,8.587,-113.070,165.601,59.809,160.744
C08530=1013.648,8.337,-113.058,165.600,59.817,160.745
C08531=1013.643,8.088,-113.045,165.598,59.826,160.746
C08532=1013.637,7.838,-113.033,165.596,59.834,160.747
C08533=1013.633,7.588,-113.020,165.593,59.842,160.748
C08534=1013.628,7.339,-113.007,165.592,59.851,160.749
C08535=1013.624,7.089,-112.995,165.589,59.859,160.750
C08536=1013.619,6.840,-112.983,165.587,59.867,160.751
C08537=1013.614,6.590,-112.970,165.584,59.876,160.752
C08538=1013.610,6.341,-112.957,165.583,59.884,160.753
C08539=1013.604,6.090,-112.944,165.581,59.893,160.754
C08540=1013.599,5.841,-112.933,165.579,59.901,160.755
C08541=1013.595,5.591,-112.920,165.577,59.909,160.756
C08542=1013.590,5.342,-112.907,165.574,59.917,160.757
C08543=1013.585,5.092,-112.895,165.572,59.925,160.758
C08544=1013.581,4.842,-112.883,165.570,59.934,160.759
C08545=1013.576,4.593,-112.870,165.568,59.942,160.760
C08546=1013.572,4.343,-112.857,165.566,59.950,160.761
C08547=1013.566,4.093,-112.845,165.563,59.958,160.762
C08548=1013.561,3.843,-112.833,165.562,59.966,160.763
C08549=1013.557,3.594,-112.820,165.560,59.974,160.764
C08550=1013.552,3.344,-112.807,165.557,59.983,160.765
C08551=1013.547,3.095,-112.795,165.555,59.991,160.766
C08552=1013.543,2.845,-112.783,165.554,59.999,160.767
C08553=1013.538,2.596,-112.770,165.551,60.007,160.768
C08554=1013.534,2.346,-112.757,165.549,60.015,160.769
C08555=1013.529,2.096,-112.746,165.547,60.023,160.770
C08556=1013.524,1.847,-112.733,165.545,60.031,160.771
C08557=1013.519,1.597,-112.720,165.543,60.039,160.772
C08558=1013.514,1.348,-112.708,165.541,60.047,160.773
C08559=1013.509,1.097,-112.696,165.539,60.055,160.774
C08560=1013.505,0.848,-112.683,165.537,60.064,160.775
C08561=1013.500,0.598,-112.670,165.534,60.071,160.776
C08562=1013.495,0.349,-112.659,165.533,60.079,160.777
C08563=1013.491,0.099,-112.646,165.531,60.087,160.778
C08564=1013.486,-0.150,-112.633,165.528,60.096,160.779
C08565=1013.482,-0.401,-112.621,165.526,60.104,160.780
C08566=1013.476,-0.650,-112.609,165.524,60.111,160.781
C08567=1013.472,-0.900,-112.597,165.522,60.119,160.782
C08568=1013.468,-1.149,-112.584,165.521,60.127,160.783
C08569=1013.462,-1.399,-112.572,165.519,60.135,160.784
C08570=1013.458,-1.649,-112.560,165.515,60.143,160.784
C08571=1013.453,-1.898,-112.547,165.514,60.151,160.785
C08572=1013.449,-2.148,-112.534,165.512,60.159,160.786
C08573=1013.444,-2.397,-112.523,165.510,60.166,160.787
C08574=1013.439,-2.647,-112.510,165.508,60.174,160.788
C08575=1013.435,-2.897,-112.498,165.506,60.181,160.789
C08576=1013.430,-3.146,-112.486,165.504,60.189,160.790
C08577=1013.425,-3.396,-112.473,165.502,60.197,160.791
C08578=1013.421,-3.646,-112.461,165.500,60.204,160.792
C08579=1013.416,-3.895,-112.448,165.497,60.213,160.793
C08580=1013.411,-4.145,-112.436,165.495,60.220,160.793
C08581=1013.407,-4.395,-112.424,165.493,60.228,160.795
C08582=1013.403,-4.645,-112.412,165.491,60.236,160.795
C08583=1013.397,-4.894,-112.399,165.489,60.244,160.796
C08584=1013.393,-5.144,-112.387,165.487,60.252,160.797
C08585=1013.388,-5.394,-112.376,165.485,60.259,160.798
C08586=1013.382,-5.670,-112.362,165.483,60.268,160.799
C08587=1013.377,-5.946,-112.350,165.480,60.277,160.800
C08588=1013.372,-6.223,-112.336,165.477,60.285,160.801
C08589=1013.367,-6.500,-112.323,165.476,60.294,160.803
C08590=1013.362,-6.749,-112.311,165.473,60.302,160.803
C08591=1013.357,-6.999,-112.300,165.471,60.310,160.804
C08592=1013.352,-7.249,-112.288,165.469,60.317,160.805
C08593=1013.347,-7.499,-112.276,165.467,60.325,160.806
C08594=1013.343,-7.748,-112.263,165.466,60.333,160.807
C08595=1013.338,-7.998,-112.252,165.463,60.340,160.808
C08596=1013.333,-8.248,-112.240,165.461,60.348,160.809
C08597=1013.329,-8.498,-112.228,165.459,60.356,160.810
C08598=1013.324,-8.746,-112.217,165.457,60.363,160.810
C08599=1013.319,-8.996,-112.205,165.455,60.371,160.811
C08600=1013.315,-9.246,-112.193,165.453,60.378,160.812
C08601=1013.310,-9.496,-112.181,165.451,60.386,160.813
C08602=1013.304,-9.745,-112.169,165.449,60.393,160.814
C08603=1013.300,-9.995,-112.157,165.446,60.401,160.815
C08604=1013.295,-10.245,-112.146,165.445,60.409,160.816
C08605=1013.290,-10.495,-112.134,165.442,60.416,160.817
C08606=1013.286,-10.744,-112.122,165.441,60.424,160.818
C08607=1013.281,-10.994,-112.110,165.438,60.431,160.818
C08608=1013.276,-11.243,-112.099,165.436,60.439,160.819
C08609=1013.272,-11.494,-112.087,165.434,60.446,160.820
C08610=1013.267,-11.743,-112.075,165.432,60.454,160.821
C08611=1013.262,-11.993,-112.063,165.430,60.461,160.822
C08612=1013.257,-12.243,-112.051,165.428,60.469,160.822
C08613=1013.253,-12.492,-112.040,165.425,60.476,160.823
C08614=1013.248,-12.742,-112.029,165.424,60.483,160.824
C08615=1013.244,-12.992,-112.017,165.422,60.491,160.825
C08616=1013.239,-13.241,-112.005,165.420,60.498,160.826
C08617=1013.233,-13.491,-111.993,165.418,60.505,160.827
C08618=1013.229,-13.741,-111.981,165.415,60.513,160.827
C08619=1013.225,-13.990,-111.970,165.413,60.520,160.828
C08620=1013.220,-14.240,-111.958,165.411,60.527,160.829
C08621=1013.215,-14.490,-111.946,165.409,60.534,160.830
C08622=1013.210,-14.740,-111.935,165.407,60.541,160.831
C08623=1013.205,-14.989,-111.923,165.405,60.549,160.831
C08624=1013.201,-15.238,-111.911,165.402,60.556,160.832
C08625=1013.196,-15.488,-111.899,165.400,60.563,160.833
C08626=1013.191,-15.738,-111.888,165.399,60.570,160.834
C08627=1013.187,-15.988,-111.876,165.397,60.578,160.834
C08628=1013.182,-16.238,-111.864,165.394,60.585,160.835
C08629=1013.178,-16.487,-111.853,165.392,60.592,160.836
C08630=1013.173,-16.737,-111.842,165.391,60.599,160.837
C08631=1013.168,-16.986,-111.830,165.389,60.607,160.838
C08632=1013.163,-17.236,-111.819,165.387,60.614,160.839
C08633=1013.159,-17.486,-111.808,165.385,60.622,160.840
C08634=1013.154,-17.736,-111.796,165.382,60.629,160.840
C08635=1013.149,-17.986,-111.785,165.381,60.636,160.841
C08636=1013.144,-18.236,-111.773,165.379,60.643,160.842
C08637=1013.140,-18.485,-111.762,165.376,60.650,160.843
C08638=1013.135,-18.735,-111.751,165.373,60.657,160.843
C08639=1013.130,-18.984,-111.739,165.372,60.664,160.844
C08640=1013.125,-19.234,-111.728,165.370,60.671,160.845
C08641=1013.121,-19.483,-111.717,165.368,60.679,160.846
C08642=1013.116,-19.734,-111.706,165.365,60.686,160.846
C08643=1013.111,-19.983,-111.695,165.364,60.693,160.847
C08644=1013.106,-20.233,-111.683,165.362,60.700,160.848
C08645=1013.101,-20.482,-111.672,165.360,60.707,160.849
C08646=1013.096,-20.732,-111.660,165.358,60.713,160.849
C08647=1013.092,-20.981,-111.649,165.355,60.721,160.850
C08648=1013.087,-21.232,-111.639,165.353,60.728,160.851
C08649=1013.082,-21.481,-111.627,165.352,60.735,160.852
C08650=1013.079,-21.695,-111.617,165.350,60.741,160.852
C08651=1013.074,-21.910,-111.607,165.347,60.746,160.853
C08652=1013.070,-22.125,-111.598,165.345,60.753,160.853
C08653=1013.066,-22.339,-111.588,165.345,60.758,160.854
C08654=1013.063,-22.554,-111.578,165.343,60.764,160.855
C08655=1013.058,-22.768,-111.569,165.341,60.770,160.855
C08656=1013.054,-22.982,-111.559,165.339,60.777,160.856
C08657=1013.051,-23.196,-111.550,165.337,60.783,160.857
C08658=1013.046,-23.446,-111.538,165.335,60.789,160.857
C08659=1013.041,-23.696,-111.527,165.333,60.796,160.858
C08660=1013.037,-23.946,-111.516,165.331,60.802,160.859
C08661=1013.032,-24.196,-111.505,165.329,60.810,160.859
C08662=1013.027,-24.445,-111.494,165.327,60.816,160.860
C08663=1013.022,-24.694,-111.482,165.324,60.823,160.861
C08664=1013.017,-24.944,-111.471,165.323,60.830,160.862
C08665=1013.013,-25.194,-111.461,165.320,60.836,160.862
C08666=1013.008,-25.444,-111.449,165.318,60.843,160.863
C08667=1013.004,-25.694,-111.437,165.317,60.849,160.864
C08668=1013.000,-25.944,-111.427,165.314,60.856,160.864
C08669=1012.995,-26.193,-111.415,165.313,60.863,160.865
C08670=1012.990,-26.443,-111.404,165.310,60.869,160.865
C08671=1012.985,-26.692,-111.393,165.309,60.876,160.866
C08672=1012.981,-26.943,-111.382,165.307,60.882,160.867
C08673=1012.976,-27.192,-111.371,165.304,60.889,160.867
C08674=1012.971,-27.442,-111.359,165.303,60.896,160.868
C08675=1012.966,-27.692,-111.348,165.300,60.902,160.869
C08676=1012.962,-27.941,-111.337,165.298,60.909,160.869
C08677=1012.957,-28.192,-111.327,165.297,60.915,160.870
C08678=1012.953,-28.441,-111.316,165.294,60.922,160.871
C08679=1012.948,-28.691,-111.305,165.292,60.928,160.871
C08680=1012.943,-28.940,-111.294,165.290,60.936,160.872
C08681=1012.938,-29.190,-111.283,165.288,60.942,160.873
C08682=1012.933,-29.440,-111.272,165.286,60.948,160.873
C08683=1012.929,-29.690,-111.262,165.284,60.955,160.874
C08684=1012.924,-29.939,-111.251,165.282,60.961,160.875
C08685=1012.920,-30.189,-111.240,165.280,60.967,160.875
C08686=1012.915,-30.439,-111.229,165.277,60.974,160.876
C08687=1012.910,-30.688,-111.219,165.276,60.981,160.877
C08688=1012.905,-30.938,-111.208,165.274,60.987,160.877
C08689=1012.901,-31.188,-111.197,165.271,60.994,160.878
C08690=1012.896,-31.438,-111.186,165.269,61.000,160.878
C08691=1012.891,-31.687,-111.176,165.267,61.006,160.879
C08692=1012.886,-31.937,-111.164,165.265,61.013,160.880
C08693=1012.882,-32.186,-111.154,165.263,61.019,160.880
C08694=1012.877,-32.437,-111.143,165.261,61.025,160.881
C08695=1012.873,-32.686,-111.132,165.259,61.032,160.882
C08696=1012.867,-32.936,-111.122,165.256,61.038,160.882
C08697=1012.863,-33.185,-111.111,165.255,61.044,160.883
C08698=1012.858,-33.436,-111.100,165.253,61.050,160.883
C08699=1012.854,-33.685,-111.090,165.251,61.057,160.884
C08700=1012.848,-33.935,-111.079,165.249,61.063,160.884
C08701=1012.844,-34.185,-111.069,165.247,61.069,160.885
C08702=1012.841,-22.372,-112.007,165.323,61.003,160.896
C08703=1012.845,-22.157,-112.017,165.325,60.998,160.896
C08704=1012.850,-21.942,-112.026,165.327,60.992,160.895
C08705=1012.853,-21.727,-112.036,165.329,60.986,160.895
C08706=1012.857,-21.512,-112.046,165.330,60.980,160.894
C08707=1012.861,-21.263,-112.057,165.333,60.974,160.894
C08708=1012.866,-21.013,-112.068,165.334,60.967,160.893
C08709=1012.871,-20.763,-112.080,165.336,60.961,160.892
C08710=1012.876,-20.514,-112.091,165.338,60.954,160.891
C08711=1012.881,-20.263,-112.102,165.340,60.947,160.891
C08712=1012.886,-20.014,-112.113,165.342,60.940,160.890
C08713=1012.890,-19.765,-112.124,165.344,60.934,160.889
C08714=1012.895,-19.515,-112.136,165.346,60.927,160.889
C08715=1012.900,-19.265,-112.147,165.348,60.920,160.888
C08716=1012.904,-19.015,-112.157,165.351,60.913,160.887
C08717=1012.909,-18.765,-112.169,165.352,60.907,160.887
C08718=1012.914,-18.516,-112.180,165.355,60.900,160.886
C08719=1012.919,-18.266,-112.192,165.356,60.893,160.885
C08720=1012.923,-18.017,-112.203,165.359,60.886,160.885
C08721=1012.928,-17.767,-112.214,165.360,60.879,160.884
C08722=1012.932,-17.516,-112.226,165.362,60.872,160.883
C08723=1012.937,-17.267,-112.237,165.364,60.866,160.882
C08724=1012.942,-17.017,-112.248,165.366,60.859,160.881
C08725=1012.947,-16.767,-112.260,165.369,60.851,160.881
C08726=1012.951,-16.518,-112.271,165.370,60.844,160.880
C08727=1012.956,-16.269,-112.282,165.373,60.838,160.879
C08728=1012.961,-16.019,-112.294,165.374,60.831,160.878
C08729=1012.965,-15.769,-112.306,165.376,60.824,160.878
C08730=1012.970,-15.519,-112.317,165.378,60.817,160.877
C08731=1012.975,-15.270,-112.329,165.380,60.810,160.876
C08732=1012.979,-15.020,-112.341,165.382,60.803,160.875
C08733=1012.984,-14.770,-112.352,165.385,60.797,160.875
C08734=1012.989,-14.520,-112.364,165.387,60.789,160.874
C08735=1012.993,-14.271,-112.375,165.388,60.783,160.873
C08736=1012.998,-14.021,-112.387,165.390,60.775,160.872
C08737=1013.003,-13.771,-112.398,165.392,60.769,160.872
C08738=1013.007,-13.521,-112.410,165.394,60.762,160.871
C08739=1013.012,-13.272,-112.422,165.397,60.754,160.870
C08740=1013.017,-13.023,-112.434,165.398,60.748,160.869
C08741=1013.021,-12.773,-112.446,165.400,60.740,160.868
C08742=1013.026,-12.523,-112.457,165.402,60.733,160.868
C08743=1013.031,-12.273,-112.469,165.404,60.726,160.867
C08744=1013.035,-12.024,-112.480,165.406,60.719,160.866
C08745=1013.040,-11.774,-112.492,165.408,60.711,160.865
C08746=1013.045,-11.524,-112.503,165.410,60.705,160.865
C08747=1013.049,-11.274,-112.516,165.412,60.698,160.864
C08748=1013.054,-11.025,-112.527,165.415,60.691,160.863
C08749=1013.059,-10.776,-112.539,165.417,60.683,160.862
C08750=1013.063,-10.525,-112.551,165.418,60.677,160.861
C08751=1013.068,-10.276,-112.562,165.420,60.668,160.860
C08752=1013.073,-10.026,-112.574,165.422,60.661,160.859
C08753=1013.078,-9.776,-112.586,165.424,60.654,160.859
C08754=1013.083,-9.527,-112.598,165.427,60.646,160.858
C08755=1013.087,-9.277,-112.609,165.428,60.640,160.857
C08756=1013.091,-9.027,-112.621,165.430,60.632,160.856
C08757=1013.096,-8.778,-112.633,165.432,60.625,160.855
C08758=1013.101,-8.528,-112.645,165.435,60.618,160.855
C08759=1013.106,-8.278,-112.657,165.436,60.610,160.854
C08760=1013.111,-8.028,-112.668,165.439,60.602,160.853
C08761=1013.115,-7.778,-112.680,165.441,60.595,160.852
C08762=1013.119,-7.529,-112.691,165.442,60.588,160.851
C08763=1013.125,-7.280,-112.704,165.444,60.580,160.850
C08764=1013.129,-7.030,-112.716,165.446,60.573,160.849
C08765=1013.134,-6.780,-112.727,165.448,60.566,160.849
C08766=1013.139,-6.530,-112.739,165.451,60.558,160.848
C08767=1013.145,-6.254,-112.752,165.453,60.550,160.847
C08768=1013.149,-5.977,-112.765,165.455,60.542,160.846
C08769=1013.154,-5.701,-112.778,165.458,60.533,160.845
C08770=1013.160,-5.425,-112.792,165.460,60.524,160.844
C08771=1013.165,-5.175,-112.803,165.462,60.517,160.843
C08772=1013.169,-4.925,-112.815,165.464,60.509,160.842
C08773=1013.174,-4.675,-112.827,165.466,60.501,160.841
C08774=1013.179,-4.426,-112.840,165.467,60.494,160.840
C08775=1013.183,-4.177,-112.851,165.469,60.487,160.839
C08776=1013.188,-3.927,-112.864,165.471,60.479,160.838
C08777=1013.192,-3.677,-112.876,165.473,60.472,160.838
C08778=1013.197,-3.428,-112.888,165.476,60.464,160.837
C08779=1013.202,-3.178,-112.900,165.477,60.456,160.836
C08780=1013.206,-2.928,-112.913,165.480,60.449,160.835
C08781=1013.211,-2.678,-112.925,165.482,60.442,160.834
C08782=1013.216,-2.429,-112.937,165.484,60.434,160.833
C08783=1013.221,-2.179,-112.950,165.486,60.426,160.832
C08784=1013.225,-1.929,-112.962,165.488,60.418,160.831
C08785=1013.229,-1.680,-112.975,165.490,60.411,160.831
C08786=1013.234,-1.430,-112.986,165.492,60.404,160.830
C08787=1013.239,-1.181,-112.999,165.494,60.396,160.829
C08788=1013.243,-0.930,-113.011,165.496,60.389,160.828
C08789=1013.248,-0.681,-113.024,165.498,60.380,160.827
C08790=1013.253,-0.432,-113.036,165.500,60.373,160.826
C08791=1013.257,-0.182,-113.048,165.502,60.365,160.825
C08792=1013.262,0.068,-113.061,165.504,60.358,160.824
C08793=1013.267,0.318,-113.072,165.506,60.350,160.823
C08794=1013.271,0.567,-113.085,165.508,60.342,160.822
C08795=1013.276,0.817,-113.098,165.510,60.335,160.821
C08796=1013.280,1.067,-113.110,165.512,60.327,160.820
C08797=1013.286,1.316,-113.122,165.514,60.319,160.819
C08798=1013.290,1.566,-113.134,165.516,60.311,160.818
C08799=1013.294,1.816,-113.147,165.517,60.303,160.817
C08800=1013.299,2.065,-113.160,165.521,60.295,160.817
C08801=1013.304,2.315,-113.171,165.522,60.287,160.816
C08802=1013.309,2.564,-113.184,165.524,60.279,160.815
C08803=1013.313,2.814,-113.197,165.526,60.271,160.813
C08804=1013.318,3.064,-113.208,165.528,60.264,160.813
C08805=1013.323,3.313,-113.221,165.530,60.256,160.812
C08806=1013.327,3.563,-113.234,165.532,60.248,160.811
C08807=1013.332,3.813,-113.246,165.534,60.240,160.810
C08808=1013.337,4.062,-113.258,165.536,60.232,160.809
C08809=1013.341,4.311,-113.271,165.538,60.224,160.808
C08810=1013.346,4.562,-113.283,165.540,60.216,160.807
C08811=1013.350,4.811,-113.296,165.543,60.208,160.806
C08812=1013.356,5.061,-113.308,165.544,60.200,160.805
C08813=1013.360,5.311,-113.320,165.546,60.192,160.804
C08814=1013.365,5.561,-113.333,165.548,60.184,160.803
C08815=1013.370,5.810,-113.345,165.550,60.175,160.802
C08816=1013.375,6.059,-113.358,165.552,60.167,160.801
C08817=1013.379,6.309,-113.370,165.554,60.159,160.800
C08818=1013.384,6.559,-113.383,165.556,60.151,160.799
C08819=1013.389,6.808,-113.395,165.558,60.143,160.798
C08820=1013.393,7.058,-113.407,165.560,60.135,160.797
C08821=1013.398,7.308,-113.420,165.563,60.126,160.796
C08822=1013.402,7.557,-113.433,165.564,60.118,160.795
C08823=1013.408,7.807,-113.445,165.566,60.110,160.794
C08824=1013.413,8.057,-113.457,165.569,60.102,160.793
C08825=1013.417,8.307,-113.470,165.570,60.094,160.792
C08826=1013.422,8.556,-113.483,165.572,60.086,160.791
C08827=1013.427,8.805,-113.495,165.575,60.077,160.790
C08828=1013.432,9.055,-113.508,165.577,60.069,160.789
C08829=1013.436,9.305,-113.520,165.579,60.061,160.788
C08830=1013.440,9.554,-113.533,165.581,60.053,160.787
C08831=1013.446,9.833,-113.547,165.583,60.043,160.785
C08832=1013.452,10.112,-113.561,165.585,60.034,160.784
C08833=1013.457,10.390,-113.575,165.588,60.024,160.783
C08834=1013.463,10.669,-113.589,165.590,60.015,160.782
C08835=1013.467,10.919,-113.601,165.592,60.007,160.781
C08836=1013.472,11.168,-113.613,165.595,59.998,160.780
C08837=1013.477,11.417,-113.626,165.596,59.990,160.778
C08838=1013.482,11.668,-113.639,165.598,59.981,160.777
C08839=1013.486,11.917,-113.652,165.600,59.973,160.776
C08840=1013.491,12.167,-113.663,165.603,59.965,160.776
C08841=1013.496,12.416,-113.676,165.604,59.956,160.774
C08842=1013.501,12.666,-113.689,165.607,59.948,160.773
C08843=1013.506,12.916,-113.702,165.609,59.938,160.772
C08844=1013.510,13.166,-113.715,165.611,59.930,160.771
C08845=1013.515,13.415,-113.728,165.612,59.923,160.770
C08846=1013.519,13.664,-113.740,165.615,59.914,160.769
C08847=1013.525,13.915,-113.754,165.616,59.905,160.768
C08848=1013.529,14.164,-113.766,165.619,59.897,160.767
C08849=1013.534,14.414,-113.779,165.621,59.889,160.766
C08850=1013.538,14.663,-113.792,165.624,59.880,160.765
C08851=1013.543,14.913,-113.805,165.625,59.872,160.763
C08852=1013.548,15.163,-113.818,165.627,59.863,160.763
C08853=1013.553,15.412,-113.831,165.629,59.855,160.761
C08854=1013.557,15.662,-113.843,165.631,59.846,160.760
C08855=1013.562,15.911,-113.857,165.633,59.838,160.759
C08856=1013.567,16.161,-113.870,165.635,59.829,160.758
C08857=1013.572,16.410,-113.883,165.637,59.821,160.757
C08858=1013.576,16.660,-113.896,165.639,59.812,160.756
C08859=1013.581,16.909,-113.908,165.642,59.803,160.755
C08860=1013.586,17.160,-113.922,165.644,59.795,160.754
C08861=1013.591,17.409,-113.934,165.646,59.786,160.753
C08862=1013.595,17.659,-113.947,165.648,59.778,160.752
C08863=1013.600,17.908,-113.960,165.650,59.769,160.750
C08864=1013.605,18.158,-113.974,165.652,59.761,160.749
C08865=1013.610,18.407,-113.987,165.654,59.752,160.748
C08866=1013.614,18.657,-113.999,165.656,59.743,160.747
C08867=1013.619,18.907,-114.013,165.658,59.735,160.746
C08868=1013.623,19.157,-114.026,165.660,59.726,160.745
C08869=1013.628,19.406,-114.039,165.662,59.718,160.744
C08870=1013.634,19.656,-114.053,165.664,59.709,160.743
C08871=1013.638,19.905,-114.065,165.667,59.700,160.742
C08872=1013.642,20.155,-114.079,165.668,59.692,160.740
C08873=1013.647,20.405,-114.092,165.671,59.683,160.739
C08874=1013.652,20.654,-114.105,165.673,59.674,160.738
C08875=1013.657,20.904,-114.118,165.675,59.666,160.737
C08876=1013.662,21.154,-114.131,165.677,59.657,160.736
C08877=1013.666,21.404,-114.145,165.678,59.648,160.735
C08878=1013.670,21.652,-114.158,165.681,59.640,160.734
C08879=1013.675,21.902,-114.171,165.683,59.631,160.733
C08880=1013.680,22.152,-114.184,165.685,59.621,160.731
C08881=1013.685,22.401,-114.198,165.687,59.614,160.730
C08882=1013.690,22.650,-114.210,165.689,59.604,160.729
C08883=1013.694,22.901,-114.224,165.692,59.595,160.728
C08884=1013.699,23.150,-114.238,165.693,59.587,160.727
C08885=1013.704,23.400,-114.251,165.696,59.578,160.726
C08886=1013.709,23.650,-114.264,165.698,59.569,160.725
C08887=1013.714,23.898,-114.277,165.700,59.560,160.723
C08888=1013.718,24.149,-114.291,165.701,59.551,160.722
C08889=1013.723,24.398,-114.304,165.704,59.543,160.721
C08890=1013.727,24.647,-114.317,165.706,59.534,160.720
C08891=1013.733,24.897,-114.330,165.708,59.524,160.719
C08892=1013.737,25.147,-114.343,165.710,59.516,160.717
C08893=1013.742,25.397,-114.357,165.712,59.507,160.716
C08894=1013.746,25.646,-114.370,165.714,59.498,160.715
C08895=1013.752,25.926,-114.385,165.717,59.488,160.714
C08896=1013.757,26.207,-114.400,165.719,59.478,160.713
C08897=1013.763,26.486,-114.415,165.722,59.468,160.711
C08898=1013.768,26.766,-114.431,165.723,59.458,160.710
C08899=1013.773,27.017,-114.444,165.725,59.449,160.709
C08900=1013.777,27.266,-114.457,165.728,59.440,160.707
C08901=1013.781,27.515,-114.471,165.730,59.431,160.706
C08902=1013.787,27.765,-114.484,165.733,59.422,160.705
C08903=1013.791,28.015,-114.498,165.734,59.413,160.704
C08904=1013.796,28.264,-114.512,165.736,59.404,160.703
C08905=1013.800,28.514,-114.525,165.739,59.395,160.702
C08906=1013.806,28.764,-114.539,165.741,59.386,160.701
C08907=1013.810,29.013,-114.552,165.742,59.377,160.699
C08908=1013.815,29.263,-114.566,165.744,59.368,160.698
C08909=1013.819,29.512,-114.579,165.747,59.359,160.697
C08910=1013.824,29.762,-114.593,165.749,59.350,160.696
C08911=1013.829,30.011,-114.607,165.751,59.341,160.695
C08912=1013.833,30.261,-114.620,165.753,59.332,160.693
C08913=1013.838,30.511,-114.634,165.755,59.323,160.692
C08914=1013.842,30.760,-114.648,165.757,59.314,160.691
C08915=1013.848,31.010,-114.662,165.759,59.305,160.690
C08916=1013.852,31.259,-114.675,165.761,59.296,160.688
C08917=1013.857,31.509,-114.689,165.764,59.287,160.687
C08918=1013.862,31.758,-114.702,165.766,59.278,160.686
C08919=1013.867,32.008,-114.717,165.768,59.269,160.685
C08920=1013.871,32.258,-114.730,165.770,59.259,160.684
C08921=1013.876,32.507,-114.744,165.772,59.251,160.682
C08922=1013.881,32.756,-114.758,165.774,59.242,160.681
C08923=1013.885,33.007,-114.771,165.776,59.233,160.680
C08924=1013.890,33.256,-114.785,165.779,59.224,160.679
C08925=1013.895,33.505,-114.799,165.780,59.214,160.677
C08926=1013.899,33.755,-114.812,165.783,59.205,160.676
C08927=1013.905,34.005,-114.826,165.785,59.196,160.675
C08928=1013.909,34.254,-114.840,165.787,59.186,160.674
C08929=1013.914,34.504,-114.853,165.789,59.177,160.673
C08930=1013.918,34.753,-114.867,165.791,59.168,160.671
C08931=1013.924,35.003,-114.881,165.793,59.158,160.670
C08932=1013.928,35.253,-114.894,165.796,59.149,160.669
C08933=1013.933,35.502,-114.908,165.798,59.140,160.668
C08934=1013.937,35.751,-114.922,165.800,59.130,160.666
C08935=1013.942,36.002,-114.936,165.802,59.121,160.665
C08936=1013.946,36.251,-114.950,165.804,59.112,160.664
C08937=1013.952,36.500,-114.964,165.807,59.103,160.663
C08938=1013.957,36.750,-114.978,165.808,59.093,160.662
C08939=1013.961,36.999,-114.992,165.811,59.084,160.660
C08940=1013.966,37.249,-115.006,165.813,59.075,160.659
C08941=1013.970,37.499,-115.019,165.815,59.066,160.658
C08942=1013.975,37.749,-115.034,165.818,59.057,160.657
C08943=1013.980,37.998,-115.047,165.819,59.047,160.655
C08944=1013.984,38.247,-115.062,165.822,59.038,160.654
C08945=1013.989,38.497,-115.076,165.824,59.029,160.653
C08946=1013.993,38.747,-115.090,165.826,59.019,160.652
C08947=1013.999,38.996,-115.104,165.828,59.010,160.651
C08948=1014.003,39.245,-115.118,165.830,59.001,160.649
C08949=1014.008,39.495,-115.133,165.833,58.992,160.648
C08950=1014.013,39.745,-115.147,165.834,58.982,160.647
C08951=1014.017,39.994,-115.161,165.837,58.973,160.646
C08952=1014.022,40.244,-115.175,165.839,58.964,160.644
C08953=1014.026,40.494,-115.188,165.841,58.954,160.643
C08954=1014.031,40.743,-115.202,165.843,58.945,160.642
C08955=1014.036,40.993,-115.217,165.845,58.936,160.640
C08956=1014.040,41.242,-115.231,165.847,58.926,160.639
C08957=1014.046,41.492,-115.245,165.850,58.917,160.638
C08958=1014.050,41.741,-115.259,165.851,58.908,160.637
